x:=1;
while (Cmd_ObjIdx <> TabDefaultLux[x].LuxNumber) and ( x <= MAX_LUXNUM) do
	x := x + 1;	
end_while
if Cmd_ObjIdx = TabDefaultLux[x].LuxNumber and TabDefaultLux[x].Mode = 2 then	// Il crono vale solo per i lux con mode = 2

(* Process command *)
CASE Cmd_C OF

	1: (* GET PROFILE *)
		IF Cmd_CLen<>3 THEN
			Cmd_R:=4;
		ELSE
			(* Load profile *)
			CronEd.CN_Sel:=WORD_TO_BYTE(Cmd_ObjIdx);
				CronEd.CN_YSel:=Cmd_Buf[9];					//**
				CronEd.CN_YSel:=shl(CronEd.CN_YSel, 8);		//**
				CronEd.CN_YSel:=CronEd.CN_YSel+Cmd_Buf[8];	//**
				//Cmd_Buf_U16:=ADR(Cmd_Buf[8]); Sostituisco questa riga e la seguente con le 3 precedenti per little/big endian (**)
				//CronEd.CN_YSel:=Cmd_Buf_U16^;
			CronEd.PR_Sel:=Cmd_Buf[10];
			CronEd.PR_Load_Exe();
				for x:=0 to 95 do
					LocalSetpoint[x]:= int_to_word(CronEd.PR.Setpoint[x]);
					LocalSetpoint[x]:=rol(LocalSetpoint[x], 8); //Scambio byte per compatibilità con sistema wago little endian
				end_for
			(* Copy data *)
			Cmd_RLen:=192;
				//TxLen:=TxLen+RAWTOHEX(ADR(CronEd.PR.Setpoint),192,ADR(TxData[TxLen]));
				TxLen:=TxLen+RAWTOHEX(ADR(LocalSetpoint),192,ADR(TxData[TxLen]));
		END_IF

	2: (* SET PROFILE *)
		IF Cmd_CLen<>(3+192) THEN
			Cmd_R:=4;
		ELSE
			(* Save profile *)
			CronEd.CN_Sel:=WORD_TO_BYTE(Cmd_ObjIdx);
				CronEd.CN_YSel:=Cmd_Buf[9];					//**
				CronEd.CN_YSel:=shl(CronEd.CN_YSel, 8);		//**
				CronEd.CN_YSel:=CronEd.CN_YSel+Cmd_Buf[8];	//**
//				Cmd_Buf_U16:=ADR(Cmd_Buf[8]); Sostituisco questa riga e la seguente con le 3 precedenti per little/big endian (**)
//				CronEd.CN_YSel:=Cmd_Buf_U16^;
			CronEd.PR_Sel:=Cmd_Buf[10];
				MEMCPY(ADR(Cmd_Buf[11]),ADR(LocalSetpoint),192); //copio i dati in locale
				for x:=0 to 95 do
					LocalSetpoint[x]:=rol(LocalSetpoint[x], 8); //Scambio byte per compatibilità con sistema wago little endian
				end_for
				MEMCPY(ADR(LocalSetpoint),ADR(CronEd.PR.Setpoint),192); //copio i byte scambiati sopra nel setpoint del crono 
//				MEMCPY(ADR(Cmd_Buf[11]),ADR(CronEd.PR.Setpoint),192);
			CronEd.PR_Save_Exe();
		END_IF

	5: (* GET CALENDAR MONTH *)
		IF Cmd_CLen<>3 THEN
			Cmd_R:=4;
		ELSE
			(* Load calendar *)
			CronEd.CN_Sel:=WORD_TO_BYTE(Cmd_ObjIdx);
				CronEd.CN_YSel:=Cmd_Buf[9];					//**
				CronEd.CN_YSel:=shl(CronEd.CN_YSel, 8);		//**
				CronEd.CN_YSel:=CronEd.CN_YSel+Cmd_Buf[8];	//**
//				Cmd_Buf_U16:=ADR(Cmd_Buf[8]); Sostituisco questa riga e la seguente con le 3 precedenti per little/big endian (**)
//				CronEd.CN_YSel:=Cmd_Buf_U16^;
			CronEd.CA_Sel:=Cmd_Buf[10];
			CronEd.CA_Load_Exe();
			(* Copy data *)
			Cmd_RLen:=32;
			TxLen:=TxLen+RAWTOHEX(ADR(CronEd.CA.Profile),32,ADR(TxData[TxLen]));
		END_IF

	6: (* SET CALENDAR MONTH *)
		IF Cmd_CLen<>(3+32) THEN
			Cmd_R:=4;
		ELSE
			(* Save calendar *)
			CronEd.CN_Sel:=WORD_TO_BYTE(Cmd_ObjIdx);
				CronEd.CN_YSel:=Cmd_Buf[9];					//**
				CronEd.CN_YSel:=shl(CronEd.CN_YSel, 8);		//**
				CronEd.CN_YSel:=CronEd.CN_YSel+Cmd_Buf[8];	//**
//				Cmd_Buf_U16:=ADR(Cmd_Buf[8]); Sostituisco questa riga e la seguente con le 3 precedenti per little/big endian (**)
//				CronEd.CN_YSel:=Cmd_Buf_U16^;
			CronEd.CA_Sel:=Cmd_Buf[10];
			MEMCPY(ADR(Cmd_Buf[11]),ADR(CronEd.CA.Profile),32);
			CronEd.CA_Save_Exe();
		END_IF
		9: (* Active crono immediatly *)
			CronEd.CN_Sel:=WORD_TO_BYTE(Cmd_ObjIdx);
			for x:= 1 to CRON_MAX do
				if CRON[x].ID = CronEd.CN_Sel then
					CRON[x].InitOK:=FALSE;
				end_if
			end_for
	else
	Cmd_R:=3;
	end_case
else 
	Cmd_R:=2;
end_if
END_ACTION

ACTION Cmd_GRU:
(* Check index *)(*
IF Cmd_ObjIdx<>1 THEN
	Cmd_R:=2;
	RETURN;
END_IF

(* Process command *)
CASE Cmd_C OF

	1: (* GET CLIMATIC *)
		Cmd_RLen:=20;
		FOR i:=0 TO 4 DO
			j:=DINT_TO_INT(GRU01_Clima.Points[i].X);
			TxLen:=TxLen+RAWTOHEX(ADR(j),2,ADR(TxData[TxLen]));
			j:=DINT_TO_INT(GRU01_Clima.Points[i].Y);
			TxLen:=TxLen+RAWTOHEX(ADR(j),2,ADR(TxData[TxLen]));
		END_FOR

	2: (* SET CLIMATIC *)
		IF Cmd_CLen<>20 THEN
			Cmd_R:=4;
		ELSE
			FOR i:=0 TO 4 DO
				Cmd_Buf_INT:=ADR(Cmd_Buf[8+4*i]); j:=Cmd_Buf_INT^;
				GRU01_Clima.Points[i].X:=INT_TO_DINT(j);
				Cmd_Buf_INT:=ADR(Cmd_Buf[10+4*i]); j:=Cmd_Buf_INT^;
				GRU01_Clima.Points[i].Y:=INT_TO_DINT(j);
			END_FOR
		END_IF

ELSE
	Cmd_R:=3;
END_CASE
*);
END_ACTION

ACTION Cmd_PDC:
(* Check index *)(*
IF Cmd_ObjIdx<>1 THEN
	Cmd_R:=2;
	RETURN;
END_IF

(* Process command *)
CASE Cmd_C OF

	3: (* TRY REARM *)
		PDC01.Rearm:=TRUE;

ELSE
	Cmd_R:=3;
END_CASE
*);
END_ACTION

ACTION Cmd_SYS:
(* Check index *)
IF Cmd_ObjIdx<>0 THEN
	Cmd_R:=2;
	RETURN;
END_IF

(* Process command *)
CASE Cmd_C OF

	0: (* ECHO *)
		IF Cmd_CLen<>0 THEN
			TxLen:=0;
		END_IF

	1: (* LOG REQUEST *)
//		LogTrig();
		(*---------------------------------------------------------------*)
			Logger_Head();
		(*---------------------------------------------------------------*)
		FOR i := 1 TO MAX_LUXNUM DO	
			if LuxElement[i].ID <> 0
			then LuxElement[i].AddLogData(WORKINGTIME:=WORKINGTIME_n[i], POWERONCYCLES:=POWERONCYCLES_n[i],
							   ENERGYCOUNTER:=ENERGYCOUNTER_n[i], ENERGYCOUNTER_T:=ENERGYCOUNTER_T_n[i]);
			end_if
		END_FOR
		(*---------------------------------------------------------------*)
			Logger_Send();
		(*---------------------------------------------------------------*)

	2: (* REARM *)
		Sys.Warning:=FALSE;
		Sys.Alarm:=FALSE;
		Sys.AlarmStop:=FALSE;

	3: (* GET INFO1 *)
		Cmd_RLen:=6;
		Plant_SN_H:= Plant_SN and 16#FFFF0000;
		Plant_SN_L:= Plant_SN and 16#0000FFFF;
		Plant_SN_H:=shr(Plant_SN_H, 16);
		Plant_SN_H_W:=dword_to_word(Plant_SN_H);
		Plant_SN_H_W:=rol(Plant_SN_H_W, 8);
		Plant_SN_L_W:=dword_to_word(Plant_SN_L);
		Plant_SN_L_W:=rol(Plant_SN_L_W, 8);
		TxLen:=TxLen+RAWTOHEX(ADR(Plant_SN_H_W),2,ADR(TxData[TxLen]));
		TxLen:=TxLen+RAWTOHEX(ADR(Plant_SN_L_W),2,ADR(TxData[TxLen]));
		//TxLen:=TxLen+RAWTOHEX(ADR(Plant_SN),4,ADR(TxData[TxLen]));
		Plant_SW_VER:=rol(Plant_SW_VER, 8);
		TxLen:=TxLen+RAWTOHEX(ADR(Plant_SW_VER),2,ADR(TxData[TxLen]));

	14: (* Set data e ora *)
		Year:=byte_to_word(Cmd_Buf[8]); 
		Year:=SHL(Year,8);
		Year:=Year + byte_to_word(Cmd_Buf[9]); 
		Year:=rol(Year, 8);
		Month:=word_to_byte(Cmd_Buf[10]); 
		Day:=word_to_byte(Cmd_Buf[12]); 
		Hour:=word_to_byte(Cmd_Buf[14]); 
		minute:=word_to_byte(Cmd_Buf[16]); 
		Sec:=word_to_byte(Cmd_Buf[18]); 
(*	
		Year:=byte_to_word(Cmd_Buf[8]); 
		Year:=SHL(Year,8);
		Year:=Year + byte_to_word(Cmd_Buf[9]); 
		Month:=word_to_byte(Cmd_Buf[11]); 
		Day:=word_to_byte(Cmd_Buf[13]); 
		Hour:=word_to_byte(Cmd_Buf[15]); 
		minute:=word_to_byte(Cmd_Buf[17]); 
		Sec:=word_to_byte(Cmd_Buf[19]); 
*)
		DTStr := concat('DT#',word_to_string(Year));
		DTStr := concat(DTStr,'-');
		DTStr := concat(DTStr,byte_to_string(Month));
		DTStr := concat(DTStr,'-');
		DTStr := concat(DTStr,byte_to_string(Day));
		DTStr := concat(DTStr,'-');
		DTStr := concat(DTStr,byte_to_string(Hour));
		DTStr := concat(DTStr,':');
		DTStr := concat(DTStr,byte_to_string(minute));
		DTStr := concat(DTStr,':');
		DTStr := concat(DTStr,byte_to_string(Sec));
		DateTime:=string_to_dt(DTStr);
		Result:=SysRtcSetTime(DateTime);
ELSE
	Cmd_R:=3;
END_CASE
END_ACTION

ACTION Command:
(* Default response OK/NODATA *)
Cmd_R:=0;
Cmd_RLen:=0;
TxLen:=16;

(* Check object *)
CASE Cmd_Obj OF

	EO_SYS:
		Cmd_SYS();
(*
	EO_GRU:
		Cmd_GRU();

	EO_PDC:
		Cmd_PDC();

	EO_CAL:
		Cmd_CAL();
*)
	EO_CRON:
		Cmd_CRON();

	EO_LUX:
		Cmd_LUX();

ELSE
	Cmd_R:=1;
END_CASE

(* Generate response *)
IF TxLen>0 THEN
	Cmd_Obj:=rol(Cmd_Obj, 8); //Scambio byte per compatibilità con sistema wago little endian
	RAWTOHEX(ADR(Cmd_Obj)	,2,ADR(TxData[ 0]));
	Cmd_ObjIdx:=rol(Cmd_ObjIdx, 8); //Scambio byte per compatibilità con sistema wago little endian
	RAWTOHEX(ADR(Cmd_ObjIdx),2,ADR(TxData[ 4]));
	Cmd_R:=rol(Cmd_R, 8); //Scambio byte per compatibilità con sistema wago little endian
	RAWTOHEX(ADR(Cmd_R)		,2,ADR(TxData[ 8]));
	Cmd_RLen:=rol(Cmd_RLen, 8); //Scambio byte per compatibilità con sistema wago little endian
	RAWTOHEX(ADR(Cmd_RLen)	,2,ADR(TxData[12]));
	TxTrig:=TRUE;
END_IF
END_ACTION

ACTION Cmd_LUX:
(* Check index *)
if Cmd_ObjIdx<1 OR Cmd_ObjIdx>MAX_LUXNUM then
	Cmd_R:=2; //id del lux fuori range
	return;
end_if

x:=1;
while (Cmd_ObjIdx <> TabDefaultLux[x].LuxNumber) and ( x <= MAX_LUXNUM) do
	x := x + 1;	
end_while
if Cmd_ObjIdx = TabDefaultLux[x].LuxNumber then	
	(* Process command *)
	case Cmd_C of
	
		0:	(* Restore default functioning mode *)
		LuxElement[x].CTRL_MODE:=LuxElement[x].CTRL_MODE_backUp;
		LuxElement[x](WORKINGTIME:=WORKINGTIME_n[x],POWERONCYCLES:=POWERONCYCLES_n[x],
													ENERGYCOUNTER:=ENERGYCOUNTER_n[x], 
													ENERGYCOUNTER_T:=ENERGYCOUNTER_T_n[x],
													CtrlExton:=KEYON);

		1:	(* Reset statistic counter *)
		LuxElement[x].StatReset(WORKINGTIME:=WORKINGTIME_n[x],POWERONCYCLES:=POWERONCYCLES_n[x],
															ENERGYCOUNTER:=ENERGYCOUNTER_n[x], 
															ENERGYCOUNTER_T:=ENERGYCOUNTER_T_n[x],
															CtrlExton:=KEYON);
	
		2,3:	(* Switch On (command=2) or Off (command=3) lux *)
		case Cmd_C of
			2: (*switch a Manuale ON*)
			LuxElement[x].CTRL_MODE := 1; // Set to manuale ON
			LuxElement[x](WORKINGTIME:=WORKINGTIME_n[x],POWERONCYCLES:=POWERONCYCLES_n[x],
														ENERGYCOUNTER:=ENERGYCOUNTER_n[x], 
														ENERGYCOUNTER_T:=ENERGYCOUNTER_T_n[x],
														CtrlExton:=KEYON);
			3: (*switch a Manuale OFF*)
			LuxElement[x].CTRL_MODE := 0; // Set to manuale OFF
			LuxElement[x](WORKINGTIME:=WORKINGTIME_n[x],POWERONCYCLES:=POWERONCYCLES_n[x],
														ENERGYCOUNTER:=ENERGYCOUNTER_n[x], 
														ENERGYCOUNTER_T:=ENERGYCOUNTER_T_n[x],
														CtrlExton:=KEYON);
			
		end_case
		4: (* Modify timer value *)
		if TabDefaultLux[x].Mode = 03 then //la modifica ha senso per i lux a timer
			NewValueTimerH:=byte_to_word(Cmd_Buf[8]);
			NewValueTimerH:=SHL(NewValueTimerH,8); 
			NewValueTimerH:=NewValueTimerH+byte_to_word(Cmd_Buf[9]);
			NewValueTimerH:=rol(NewValueTimerH, 8);

			NewValueTimerL:=byte_to_word(Cmd_Buf[10]);
			NewValueTimerL:=SHL(NewValueTimerL,8); 
			NewValueTimerL:=NewValueTimerL+byte_to_word(Cmd_Buf[11]);
			NewValueTimerL:=rol(NewValueTimerL, 8);
			
			NewValueTimer:=word_to_dword(NewValueTimerH);			
			NewValueTimer:=SHL(NewValueTimer,16);
			NewValueTimer:=NewValueTimer+word_to_dword(NewValueTimerL);
			if NewValueTimer>4294966 then
				Cmd_R:=3; //Comando errato valore timer overflow		
			
(*
			NewValueTimer:=byte_to_dword(Cmd_Buf[8]);
			NewValueTimer:=SHL(NewValueTimer,8); 
			NewValueTimer:=NewValueTimer+byte_to_dword(Cmd_Buf[9]);
			NewValueTimer:=SHL(NewValueTimer,8); 
			NewValueTimer:=NewValueTimer+byte_to_dword(Cmd_Buf[10]);
			NewValueTimer:=SHL(NewValueTimer,8); 
			NewValueTimer:=NewValueTimer+byte_to_dword(Cmd_Buf[11]);
*)
			else
					TabLuxPsg[x].TimerOn := dword_to_time(NewValueTimer*1000);
				for x := 1 to MAX_LUXNUM do
					if LuxElement[x].ID = Cmd_ObjIdx
						then LuxElement[x].LuxTimer := dword_to_time(NewValueTimer*1000); //set del nuovo valore del timer del lux 	
					end_if
				end_for
			end_if
		else
			Cmd_R:=3; //Comando errato / non previsto
		end_if
		5:	(* get working mode*)
			Cmd_RLen:=2;
			ModeFromPlc:=LuxElement[x].CTRL_MODE;
			ModeFromPlc:=rol(ModeFromPlc, 8);
			TxLen:=TxLen+RAWTOHEX(ADR(ModeFromPlc),2,ADR(TxData[TxLen]));
//		6: (* Modify dimming value for timer control *)
//		7: (* Modify dimming value for key control *)
//		8: (* Modify start and stop orari di funzionamento dei lux a timer *)
	else
		Cmd_R:=3; //Comando errato / non previsto
	end_case
else
	Cmd_R:=2; //id del lux non presente in lista
end_if
END_ACTION

END_PROGRAM

// Utils Functions/HEXTORAW
FUNCTION HEXTORAW : WORD
VAR_INPUT
	pString		: POINTER TO BYTE;
	StringLen	: WORD;
	pData		: POINTER TO BYTE;
END_VAR
VAR
	xl: WORD;
	xi: WORD;
	xr: BYTE;
END_VAR

xl:=0;
xi:=0;

WHILE xi<StringLen DO

	IF pString^>=97 AND pString^<=102 THEN
		xr := pString^ - 87;
	ELSIF pString^>=65 AND pString^<=70 THEN
		xr := pString^ - 55;
	ELSIF pString^>=48 AND pString^<=57 THEN
		xr := pString^ - 48;
	ELSE
		xr := 16;
	END_IF

	IF xr<16 THEN
		IF (xi AND 1)=0 THEN
			pData^ := xr * 16;
		ELSE
			pData^ := pData^ + xr;
			pData := pData + 1;
			xl := xl + 1;
		END_IF
	END_IF

	xi := xi + 1;
	pString := pString + 1;

END_WHILE

HEXTORAW:=xl;

END_FUNCTION

// Utils Functions/TCPSERVER
FUNCTION_BLOCK TCPSERVER
(***********************************************************************************************************	*)
(* Version: 1.6                                    			          											*)
(* Date: 11.02.2011                                   					          							    *)
(***********************************************************************************************************	*)
(* WAGO Kontakttechnik GmbH Hansastr. 27 32423 Minden(Westf.)													*)
(* Tel. +0049 571/887-0 Fax. +0049 571/887-0																	*)
(* Author: VB																									*)
(***********************************************************************************************************	*)
(*Description:	A TCP server to read and write data													       		*)
(*Historie:																										*)
(*Version 1.6: 11.02.2011: Changes according to 750-880/881											 			*)
(*Version 1.5: 27.11.2008 Bugfix allow reuse port																*)
(*Version 1.4: 13.10.2008 Bugfix transmitting large data														*)
(*Version 1.3: 15.01.2007 Changes according to FW11																*)
(*Version 1.2: 09.03.2006 Changes for socket handle 0											       			*)
(*Version 1.1: 14.02.2005 Release																				*)
(***********************************************************************************************************	*)
VAR CONSTANT
	STATE_INIT     				 : BYTE:= 0;
	STATE_OPEN     				 : BYTE:= 1;
	STATE_TX       				 : BYTE:= 20;
	STATE_RX       				 : BYTE:= 30;
	STATE_CLOSE    				 : BYTE:= 40;
	STATE_ERROR_TRAP		 	 : BYTE:= 200;
END_VAR
VAR_INPUT
	xEnable    					: BOOL;	 (* Set TRUE to enable function block *)
	wPortNumber					: WORD;  (* Port *)
	tServerTimeOut				: TIME:=t#50s;
	ptSendData					: POINTER TO ARRAY[0..MAX_SEND_TCP_SERVER] OF BYTE;
	diSendCount					: DINT;
END_VAR
VAR_OUTPUT
	xClientConnected  			: BOOL:= FALSE;
	diError 					: DINT:= 0;
END_VAR
(* Status Codes -----------------------------------------
	16#8001 => No socket descriptor available 
	16#8002 => SysSockBind fails 
	16#8003 => SysSockListen fails 
	16#8004 => switching to none blocking mode fails
	16#8005 => SysSockClose() returns FALSE 
    16#8006 => SysSockConnect() fails
    16#8007 => SysSockSend() fails
	16#8008 => error state machine 
	16#8009 => timeout while waiting for data from server 
	16#0001 => server waiting for client to establish connection
------------------------------------------------------------*)
VAR_IN_OUT
	xStartSend					: BOOL;
	aReceiveBuffer				: ARRAY [0..MAX_RECEIVE_TCP_SERVER] OF BYTE;
	diReceiveCount				: DINT;
END_VAR

VAR
	m_State    					: BYTE:= 0;
	m_ReceiveBuffer				: ARRAY [0..MAX_RECEIVE_TCP_SERVER_SOCKET] OF BYTE;
	m_ServerSocket				: DINT:= SOCKET_INVALID;
	m_Socket					: DINT:= SOCKET_INVALID;
	m_AddressInfo				: SOCKADDRESS;
	m_BytesReceived				: DINT;
	m_diReturn					: DINT;
	m_xReturn					: BOOL;
	m_SizeSockadr				: DWORD;
	m_ConnectionWatchdog		: TON;
	m_Flags						: DINT;
	m_NoneBlocking   			: DINT:= 1;
	m_Blocking   				: DINT:= 0;
	i							: INT;
	m_count						: DINT;
	diOption					: DINT := 1;
	on: DINT;
	errorCode					: DINT;
	errorCodeLenght				: dint;
	xResultErrCode				: bool;
END_VAR

IF xEnable THEN
	CASE m_State OF
		STATE_INIT:
			(* Create Socket *)
			m_ServerSocket:= SysSockCreate( SOCKET_AF_INET, SOCKET_STREAM, 0);
			IF m_ServerSocket = SOCKET_INVALID THEN
				(* *)
				diError:= 16#8001;
				m_State:= STATE_ERROR_TRAP;
				RETURN;
			ELSE
				;
			END_IF
			(* Address bindings *)
			(********************)
			on:=1;
			SysSockSetOption( m_ServerSocket, SOCKET_SOL, SOCKET_SO_REUSEADDR, ADR(on), SIZEOF(on) );

			m_AddressInfo.sin_family:= SOCKET_AF_INET;
			m_AddressInfo.sin_port  := SysSockHtons( wPortNumber);
			m_AddressInfo.sin_addr  := SOCKET_INADDR_ANY;
			IF NOT SysSockBind( m_ServerSocket, ADR(m_AddressInfo), SIZEOF(m_AddressInfo)) THEN
				diError:= 16#8002;
				m_State:= STATE_ERROR_TRAP;
				RETURN;
			END_IF
			(* Wait for connections *)
			(************************)
			IF NOT SysSockListen( m_ServerSocket, 1) THEN
				diError:= 16#8003;
				m_State:= STATE_ERROR_TRAP;
			END_IF

			(* Puts SOCKET in NonBlocking mode *)
			m_diReturn:= SysSockIoctl( m_ServerSocket, SOCKET_FIONBIO, ADR(m_NoneBlocking));

			m_State:= STATE_OPEN;


		STATE_OPEN: 	(* Waiting for incomming connection *)
				m_SizeSockadr:=SIZEOF(m_AddressInfo);
				m_Socket:= SysSockAccept( m_ServerSocket, ADR(m_AddressInfo), ADR(m_SizeSockadr));
				diError:=State_open;
				IF m_Socket <> SOCKET_INVALID THEN
					xClientConnected:=TRUE;
					(*Set Push-Bit:new V1.5*)
				(*	IF ADR(%MW0)=16#30000000  OR ADR(%MW0)=16#20000000 THEN (*841 or 881*)
						SysSockSetOption(
							diSocket:=m_Socket,
							diLevel:=6,
							diOption:=SOCKET_TCP_NODELAY,
							pOptionValue:=ADR(diOption),
							diOptionLength:=SIZEOF(diOption));
					ELSE
							;
					END_IF *)
					SysSockIoctl( m_Socket, SOCKET_FIONBIO, ADR(m_NoneBlocking));
					m_State:= STATE_RX;
					diError:=0;
				END_IF

		STATE_RX:
					errorCodeLenght:=sizeof(errorCode);
					xResultErrCode:=SysSockGetOption(m_Socket,  SOCKET_SOL, SOCKET_SO_KEEPALIVE, adr(errorCode), adr(errorCodeLenght));
					m_BytesReceived:= SysSockRecv( m_Socket, ADR(m_ReceiveBuffer), SIZEOF(m_ReceiveBuffer), 0);
					CASE m_BytesReceived OF
					-1:(*no data available or error occured*)
						m_ConnectionWatchdog(IN:=TRUE , PT:=T#200ms);	//tServerTimeOut );
						IF m_connectionWatchdog.Q THEN
							m_State:= STATE_CLOSE;
							m_ConnectionWatchdog(IN:=FALSE);(*reset connection watchdog*)
							diError := 16#8009;
						END_IF
					0:(* socket was "gracefully closed"  *)
						m_State:= STATE_CLOSE;
						diError := 16#8003;
					ELSE
						(* Copy received data into receive buffer *)
						(********************************)
						FOR i:= 0 TO DINT_TO_INT(m_BytesReceived	)-1 DO
							aReceiveBuffer[diReceiveCount]:= m_ReceiveBuffer[i];
							diReceiveCount:=(diReceiveCount+1) MOD SIZEOF(aReceiveBuffer);
						END_FOR

						m_ConnectionWatchdog(IN:=FALSE);(*reset connection watchdog*)
					END_CASE

				(*send data*)
				IF xStartSend	 THEN
					m_State := STATE_TX;
				END_IF

	STATE_TX:	 (* send TCP-message *)
		m_diReturn := SysSockSend(diSocket := m_Socket,
								  pbyBuffer := ADR(ptSendData^[m_count]),(*geändert V1.4 bisher: [0] *)
								  diBufferSize := diSendCount-m_count,
								  diFlags :=m_Flags);
		CASE m_diReturn OF
		-1:	(* ERROR or data could not yet be send (V1.3 due to new FW11) *)
			m_ConnectionWatchdog(IN:=TRUE , PT:=tServerTimeOut );
			IF m_connectionWatchdog.Q THEN
				m_State:= STATE_CLOSE;
				m_ConnectionWatchdog(IN:=FALSE);(*reset connection watchdog*)
				diError := 16#8007;
			END_IF
		0: (* socket was "gracefully closed"  *)
			m_State := STATE_CLOSE;
			diError := 16#8003;
		ELSE (* succesful *)
			m_count:=m_count+m_diReturn;
			IF m_count>=diSendCount THEN
				diError := 16#0000;
				m_State := STATE_RX;
				m_count:=0;
				xStartSend:=FALSE;
			END_IF
			m_ConnectionWatchdog(IN:=FALSE);(*reset connection watchdog*)
		END_CASE


		STATE_CLOSE:	(* Close the server *)

	(*	IF ADR(%MW0)=16#30000000  OR ADR(%MW0)=16#20000000 THEN (*841 or 881*)
			;
		ELSE
			IF m_Socket>=0 THEN
				SysSockShutdown(m_Socket, 0);;(*870*)
			END_IF
		END_IF  *)
		IF m_Socket>=0 THEN
			SysSockClose( m_Socket);
		END_IF
		xClientConnected:= FALSE;
		m_State:= STATE_OPEN; (* Try to open the server again *)
		m_ConnectionWatchdog(IN:=FALSE);(*reset connection watchdog*)

		STATE_ERROR_TRAP: (* Error Read/Write socket  *)
			m_State:= STATE_ERROR_TRAP;

	ELSE  (* Bad FSM code trap  *)
			m_State:= STATE_ERROR_TRAP;
			diError:= 16#8008;
	END_CASE;
ELSE
	IF m_State <> STATE_INIT THEN
	(*	IF ADR(%MW0)=16#30000000  OR ADR(%MW0)=16#20000000 THEN (*841 or 881*)
			;
		ELSE
			IF m_Socket>=0 THEN
				SysSockShutdown(m_Socket, 0);;(*870*)
			END_IF
		END_IF *)
		IF m_Socket>=0 THEN
			SysSockClose( m_Socket);
		END_IF
	(*	IF ADR(%MW0)=16#30000000  OR ADR(%MW0)=16#20000000 THEN (*841 or 881*)
			;
		ELSE
			IF m_ServerSocket>=0 THEN
				SysSockShutdown(m_ServerSocket, 0);;(*870*)
			END_IF
		END_IF  *)
		IF m_ServerSocket>=0 THEN
			SysSockClose( m_ServerSocket);
		END_IF
		xClientConnected:= FALSE;
		diError:= 0;
		m_State:= STATE_init; (* Try to open the server again *)
		m_ConnectionWatchdog(IN:=FALSE);(*reset connection watchdog*)
	END_IF
END_IF

END_FUNCTION_BLOCK

// Utils Functions/RAWTOHEX
FUNCTION RAWTOHEX : WORD
VAR_INPUT
	pData: POINTER TO BYTE;
	DataLen: WORD;
	pString: POINTER TO BYTE;
END_VAR
VAR
	xl: WORD;
END_VAR

xl:=0;

WHILE DataLen>0 DO

	pString^ := (pData^ / 16#10) + 48 + (((pData^ / 16#10)/10)*7);
	pString:=pString+1;
	pString^ := (pData^ AND 16#0F)  + 48 + (((pData^ AND 16#0F)/10)*7);
	pString:=pString+1;
	pData:=pData+1;
	DataLen:=DataLen-1;
	xl:=xl+2;

END_WHILE

(*pString^:=0;*)

RAWTOHEX:=xl;

END_FUNCTION

// TCP_Logger/LogTrig
FUNCTION LogTrig : BOOL
VAR
	s1 		: STRING(255);	//STRING(160);
	i, j, k	: word;
END_VAR

(*---------------------------------------------------------------*)
	Logger_Head();
(*---------------------------------------------------------------*)
case enSelect of
	Sel_PSG: (* Log PSG *)

for i := 1 TO PSG_MAXNUM DO	
	if PSG[i].ID <> 0
	then PSG[i].AddLogData(NumTransition:=PsgCounter[i]);	//PSG[i].AddLogData(NumTransition:=PsgCounter[PSG[i].ID]);
 	end_if
END_FOR
		enSelect:=Sel_LUX;
		
	Sel_LUX: (* Log LUXM *)
		
FOR i := 1 TO MAX_LUXNUM DO	
	if LuxElement[i].ID <> 0
	then LuxElement[i].AddLogData(WORKINGTIME:=WORKINGTIME_n[i], POWERONCYCLES:=POWERONCYCLES_n[i],
					   ENERGYCOUNTER:=ENERGYCOUNTER_n[i], ENERGYCOUNTER_T:=ENERGYCOUNTER_T_n[i]);
 	end_if
END_FOR
		enSelect:=Sel_CRON;
	Sel_CRON: (* Log CRON *)

FOR i := 1 TO CRON_MAX DO
	if CRON[i].ID <> 0
		then CRON[i].AddLogData(SET_POINT:=CRON[i].SetPoint, STAT_LOG:=CRON[i].Status_Log);
	end_if
END_FOR

		enSelect:=Sel_END;
END_CASE
(* Log LUXM *)
	(* 
FOR i := 1 TO MAX_LUXNUM DO	
	if LuxElement[i].ID <> 0
	then LuxElement[i].AddLogData(WORKINGTIME:=WORKINGTIME_n[i], POWERONCYCLES:=POWERONCYCLES_n[i],
					   ENERGYCOUNTER:=ENERGYCOUNTER_n[i], ENERGYCOUNTER_T:=ENERGYCOUNTER_T_n[i]);
 	end_if
END_FOR
 *)

(*---------------------------------------------------------------*)
	Logger_Send();
(*---------------------------------------------------------------*)

END_FUNCTION

// Utils Functions/TestAsi_FB
FUNCTION_BLOCK TestAsi_FB
VAR_INPUT
END_VAR
VAR_OUTPUT
END_VAR
VAR
	TTestOut: tof
;
	iCounter0: INT := 0;
	TrigH:	BOOL;
	rTrigger: R_TRIG;
END_VAR

(*
TTestOut(IN:=NOT TTestOut.Q,PT:=T#5S);
IF TTestOut.Q AND LUXM_46 = FALSE
THEN
	LUXM_46:=TRUE;	
	ELSE
		IF NOT TTestOut.Q
			THEN
				LUXM_46 := FALSE;
		END_IF
END_IF
IF 	LUXST_46 THEN
	IF iCounter0 < 65535 THEN
		iCounter0:=iCounter0+1;	
	END_IF
END_IF
*)
//rTrigger(CLK:=PSG89_IN);
//TTestOut(IN:=NOT PSG89_IN ,PT:=T#5S);
//IF rTrigger.q THEN
 	//TTestOut(IN:=rTrigger.q ,PT:=T#5S);
//END_IF
(*
IF TTestOut.Q THEN 
	LUXM_46:=TRUE;	
	ELSE
		LUXM_46:=FALSE;	
END_IF
*)
(*
IF 	Asi_in0901 THEN
	IF iCounter1 < 65535 THEN
		iCounter1:=iCounter1+1;	
	END_IF

END_IF

IF 	Asi_in0902 THEN
	IF iCounter2 < 65535 THEN
		iCounter2:=iCounter2+1;	
	END_IF
END_IF

IF 	Asi_in0903 THEN
	IF iCounter3 < 65535 THEN
		iCounter3:=iCounter3+1;	
	END_IF

END_IF
*)

END_FUNCTION_BLOCK

// Utils Functions/OpenFiles_ASI_PSG_FB
//Esegue la lettura del file x_ASI_PSG.txt per poi configurare le tabelle ASI_1 e ASI_2 di associazione tra passaggi e segnali di input 
FUNCTION_BLOCK OpenFiles_ASI_PSG_FB
VAR_INPUT
	//sFileName : STRING;
END_VAR
VAR_OUTPUT
	Message		: STRING;
END_VAR
VAR
	hMode		: ACCESS_MODE;
	hFile		: RTS_IEC_HANDLE;
	hRes		: RTS_IEC_RESULT;
	bList		: ARRAY [0..15] OF BYTE;
	i			: DWORD; //Dim max file: 2^32 byte
	j			: BYTE; //Indice dell'array bList
	k			: BYTE; //Indice tabella ASI 2^8 = 256
	xwDimFile	: LWORD;
	bChar		: BYTE;
	sFileName 	: STRING;
END_VAR

(* Create current filename 'yyyyCRnn.DAT' *)
//sFileName:=CONCAT(ConfPath,WORD_TO_STRING('2ASI_LUX.txt'));
//sFileName:=CONCAT(STR1:=sFileName, STR2:='CR');
//IF CN_Sel<10 THEN
//sFileName:=CONCAT(STR1:=sFileName, STR2:='0');
//END_IF
//sFileName:=CONCAT(STR1:=sFileName, STR2:=BYTE_TO_STRING(CN_Sel));
//sFileName:=CONCAT(STR1:=sFileName, STR2:='.DAT');
//sFileName:='/media/sd/2015CR01.DAT';	//2_ASI_LUX.txt';
(* Check file version and size! *)
(* ... *)
Message:='';
(* Open data file *)
sFileName:=CONCAT(STR1:=MapConf_Path, STR2:=PLC_ID);
sFileName:=CONCAT(STR1:=sFileName, STR2:=AsiPsg_FileName);
hFile:=SysFileOpen(sFileName,AM_READ,ADR(hRes));

(* File not found *)
IF hFile=RTS_INVALID_HANDLE THEN
	Message:='File not found';
	RETURN;
END_IF

(* Close file *)
SysFileClose(hFile);

(* Open data file *)
i:=0; //indice di scorrimento del file
j:=0; //indice di scorrimento dell'array dove viene momentaneamente memorizzata la riga prima del ;
k:=0; //indice della tabella di mappatura ASI
hFile:=SysFileOpen(sFileName,hMode,ADR(hRes));
//-------------- MODIFICA START --------------------
	SysFileSetPos(hFile, i);	
	SysFileRead(hFile, ADR(bList[j]), 1, ADR(hRes));
//-------------- MODIFICA END --------------------
WHILE SysFileEOF(hFile)<> 0 DO
//	SysFileSetPos(hFile, i);	
//	SysFileRead(hFile, ADR(bList[j]), 1, ADR(hRes));
	IF bList[j] = 16#2F  // se trovo '/'
		THEN 
			SysFileSetPos(hFile, i+1);	
			SysFileRead(hFile, ADR(bList[j+1]), 1, ADR(hRes));
			IF bList[j+1] = 16#2F  // se trovo ancora '/'
				THEN 
					WHILE  bList[j]<> 16#0D DO
						i := i+1;
						SysFileSetPos(hFile, i);	
						SysFileRead(hFile, ADR(bList[j]), 1, ADR(hRes));
					END_WHILE	
					i := i+1;
					SysFileSetPos(hFile, i);	
					SysFileRead(hFile, ADR(bList[j]), 1, ADR(hRes));
					IF bList[j] = 16#0A
						THEN 
							i := i+1;
							j := 0;
							SysFileSetPos(hFile, i);	
							SysFileRead(hFile, ADR(bList[j]), 1, ADR(hRes)); //leggo il primo carattere della nuova riga
						ELSE 
							Message:='Errore 0D 0A';
							RETURN;
					END_IF
				ELSE 
					Message:='Errore //';
					RETURN;
			END_IF
	END_IF
	IF bList[j] <> 16#3B //finchè non trovo ;
		THEN 
			i:=i+1;
			j:=j+1;	
		ELSE
			i:=i+3; //Se trovo ; inizio a salvare i dati della riga letta in TabAsiPsg[k]....
			j:=0;
			k:=k+1;
			TabAsiPsg[k].Asi1_2 := (bList[0]-16#30); //memorizzo se asi 1 o asi 2
			IF 	bList[4] = 16#41	//Se contiene il carattere A
				THEN TabAsiPsg[k].A_B := ASI_A;
				ELSE TabAsiPsg[k].A_B := ASI_B;
			END_IF	
			TabAsiPsg[k].Address :=  (bList[2]-16#30)*10 + (bList[3]-16#30); //memorizzo indirizzo
			TabAsiPsg[k].bit_psg[bList[6]-16#30] := (bList[8]-16#30)*100 + (bList[9]-16#30)*10 + (bList[10]-16#30); //memorizzo il passaggio associato 
			//TabAsiPsg[k].PSG := (bList[8]-16#30)*100 + (bList[9]-16#30)*10 + (bList[10]-16#30); //memorizzo il passaggio associato
			IF 	(k> 1) AND (TabAsiPsg[k].Asi1_2 = TabAsiPsg[k-1].Asi1_2) AND (TabAsiPsg[k].A_B = TabAsiPsg[k-1].A_B) AND (TabAsiPsg[k].Address = TabAsiPsg[k-1].Address)
				THEN //memorizzo il passaggio associato nella struttura k-1 perchè di uguale indirizzo
					TabAsiPsg[k-1].bit_psg[bList[6]-16#30] := (bList[8]-16#30)*100 + (bList[9]-16#30)*10 + (bList[10]-16#30);  
					TabAsiPsg[k].Asi1_2 := 0;	//pulisco l'array
					TabAsiPsg[k].A_B := 0;	//pulisco l'array
					TabAsiPsg[k].Address := 0;	//pulisco l'array
					TabAsiPsg[k].bit_psg[bList[6]-16#30] := 0;	//pulisco l'array
					k := k-1;	//riposiziono il contatore
			END_IF
			(*		
			CASE bList[0] OF
			16#31:
				IF 	bList[4] = 16#41	//Se contiene il carattere A
					THEN TabASI1[k].A_B := ASI_A;
					ELSE TabASI1[k].A_B := ASI_B;
				END_IF		
				TabASI1[k].Address :=  (bList[2]-16#30)*10 + (bList[3]-16#30);
				TabASI1[k].Bit_address := bList[6]-16#30;
				TabASI1[k].PSG := (bList[8]-16#30)*100 + (bList[9]-16#30)*10 + (bList[10]-16#30);
				
			16#32:
				IF 	bList[4] = 16#41	//Se contiene il carattere A
					THEN TabASI2[k].A_B := ASI_A;
					ELSE TabASI2[k].A_B := ASI_B;
				END_IF		
				TabASI2[k].Address :=  (bList[2]-16#30)*10 + (bList[3]-16#30);
				TabASI2[k].Bit_address := bList[6]-16#30;
				TabASI2[k].PSG := (bList[8]-16#30)*100 + (bList[9]-16#30)*10 + (bList[10]-16#30);
		END_CASE 
			CASE bList[0] OF
			16#31:
				IF 	bList[4] = 16#41	//Se contiene il carattere A
					THEN TabASI1AB_FromFile[1] := ASI_A;
					ELSE TabASI1AB_FromFile[1] := ASI_B;
				END_IF		
				TabASI1Add_FromFile[1] :=  (bList[2]-16#30)*10 + (bList[3]-16#30);
				TabASI1BitAdd_FromFile[1] := bList[6]-16#30;
				TabASI1PSG_FromFile[1] := (bList[8]-16#30)*100 + (bList[9]-16#30)*10 + (bList[10]-16#30);
			16#32:
				IF 	bList[4] = 16#41	//Se contiene il carattere A
					THEN TabASI2AB_FromFile[1] := ASI_A;
					ELSE TabASI2AB_FromFile[1] := ASI_B;
				END_IF		
				TabASI2Add_FromFile[1] :=  (bList[2]-16#30)*10 + (bList[3]-16#30);
				TabASI2BitAdd_FromFile[1] := bList[6]-16#30;
				TabASI2PSG_FromFile[1] := (bList[8]-16#30)*100 + (bList[9]-16#30)*10 + (bList[10]-16#30);
		END_CASE *)
	END_IF	
//-------------- MODIFICA START --------------------
	SysFileSetPos(hFile, i);	
	SysFileRead(hFile, ADR(bList[j]), 1, ADR(hRes));
//-------------- MODIFICA END --------------------
END_WHILE
if SysFileEOF(hFile) = 0 
	then Message:='Reading ASI_Psg File: OK';
end_if
//xwDimFile:=SysFileGetSize(sFileName,ADR(hRes));
(* Close file *)
SysFileClose(hFile);

END_FUNCTION_BLOCK

// Utils Functions/OpenFiles_ASI_LUX_FB
//Esegue la lettura del file x_ASI_LUX.txt per poi configurare le tabelle ASI_1 e ASI_2 di associazione tra LUX e segnali di output 
FUNCTION_BLOCK OpenFiles_ASI_LUX_FB
VAR_INPUT
END_VAR
VAR_OUTPUT
	Message		: STRING;
END_VAR
VAR
	hMode		: ACCESS_MODE;
	hFile		: RTS_IEC_HANDLE;
	hRes		: RTS_IEC_RESULT;
	bList		: ARRAY [0..15] OF BYTE;
	i			: DWORD;
	j			: DWORD;
	k			: byte;
	xwDimFile	: LWORD;
	bChar		: BYTE;
	sFileName 	: STRING;
END_VAR

Message:='';
(* Open data file *)
sFileName:=CONCAT(STR1:=MapConf_Path, STR2:=PLC_ID);
sFileName:=CONCAT(STR1:=sFileName, STR2:=AsiLux_FileName);
hFile:=SysFileOpen(sFileName,AM_READ,ADR(hRes));

(* File not found *)
IF hFile=RTS_INVALID_HANDLE THEN
	Message:='File not found';
	RETURN;
END_IF

(* Close file *)
SysFileClose(hFile);

(* Open data file *)
i:=0;
j:=0;
k:=0;
hFile:=SysFileOpen(sFileName,hMode,ADR(hRes));
//-------------- MODIFICA START --------------------
	SysFileSetPos(hFile, i);	
	SysFileRead(hFile, ADR(bList[j]), 1, ADR(hRes));
//-------------- MODIFICA END --------------------
WHILE SysFileEOF(hFile)<> 0 DO
//	SysFileSetPos(hFile, i);	
//	SysFileRead(hFile, ADR(bList[j]), 1, ADR(hRes));
	IF bList[j] = 16#2F  // se trovo '/'
		THEN 
			SysFileSetPos(hFile, i+1);	
			SysFileRead(hFile, ADR(bList[j+1]), 1, ADR(hRes));
			IF bList[j+1] = 16#2F  // se trovo ancora '/'
				THEN 
					WHILE  bList[j]<> 16#0D DO
						i := i+1;
						SysFileSetPos(hFile, i);	
						SysFileRead(hFile, ADR(bList[j]), 1, ADR(hRes));
					END_WHILE	
					i := i+1;
					SysFileSetPos(hFile, i);	
					SysFileRead(hFile, ADR(bList[j]), 1, ADR(hRes));
					IF bList[j] = 16#0A
						THEN 
							i := i+1;
							j := 0;
							SysFileSetPos(hFile, i);	
							SysFileRead(hFile, ADR(bList[j]), 1, ADR(hRes)); //leggo il primo carattere della nuova riga
						ELSE 
							Message:='Errore 0D 0A';
							RETURN;
					END_IF
				ELSE 
					Message:='Errore //';
					RETURN;
			END_IF
	END_IF
	IF bList[j] <> 16#3B //finchè non trovo ;
		THEN 
			i:=i+1;
			j:=j+1;	
		ELSE
			i:=i+3; //Se trovo ; inizio a salvare i dati della riga letta in TabASILux[k]....
			j:=0;
			k:=k+1;
			TabASILux[k].Asi1_2 := (bList[0]-16#30); //memorizzo se asi 1 o asi 2
			IF 	bList[4] = 16#41	//Se contiene il carattere A
				THEN TabASILux[k].A_B := ASI_A;
				ELSE TabASILux[k].A_B := ASI_B;
			END_IF		
			TabASILux[k].Address :=  (bList[2]-16#30)*10 + (bList[3]-16#30); //memorizzo indirizzo
			TabASILux[k].bit_lux[bList[6]-16#30] := (bList[8]-16#30)*100 + (bList[9]-16#30)*10 + (bList[10]-16#30); //memorizzo il lux associato 
			IF 	(k> 1) AND (TabASILux[k].Asi1_2 = TabASILux[k-1].Asi1_2) AND (TabASILux[k].A_B = TabASILux[k-1].A_B) AND (TabASILux[k].Address = TabASILux[k-1].Address)
				THEN //memorizzo il passaggio associato nella struttura k-1 perchè di uguale indirizzo
					TabASILux[k-1].bit_lux[bList[6]-16#30] := (bList[8]-16#30)*100 + (bList[9]-16#30)*10 + (bList[10]-16#30);  
					TabASILux[k].Asi1_2 := 0;	//pulisco l'array
					TabASILux[k].A_B := 0;	//pulisco l'array
					TabASILux[k].Address := 0;	//pulisco l'array
					TabASILux[k].bit_lux[bList[6]-16#30] := 0;	//pulisco l'array
					k := k-1;	//riposiziono il contatore
			END_IF
			
//			TabASILux[k].Address :=  (bList[2]-16#30)*10 + (bList[3]-16#30); //memorizzo indirizzo
//			TabASILux[k].Bit_address := bList[6]-16#30;		//memorizzo il bit
//			TabASILux[k].LUX := (bList[8]-16#30)*100 + (bList[9]-16#30)*10 + (bList[10]-16#30); //memorizzo il passaggio associato
	END_IF	
//-------------- MODIFICA START --------------------
	SysFileSetPos(hFile, i);	
	SysFileRead(hFile, ADR(bList[j]), 1, ADR(hRes));
//-------------- MODIFICA END --------------------
END_WHILE
if SysFileEOF(hFile) = 0 
	then Message:='Reading ASI_Lux File: OK';
end_if
(* Close file *)
SysFileClose(hFile);

END_FUNCTION_BLOCK

// Utils Functions/OpenFiles_LUX_PSG_FB
//Esegue la lettura del file x_AUT_LUX_PSG.txt per poi configurare le associazione tra passaggi e lux corrispondenti
FUNCTION_BLOCK OpenFiles_LUX_PSG_FB
VAR_INPUT
	//sFileName : STRING;
END_VAR
VAR_OUTPUT
	Message		: STRING;
END_VAR
VAR
	hMode		: ACCESS_MODE;
	hFile		: RTS_IEC_HANDLE;
	hRes		: RTS_IEC_RESULT;
	bList		: ARRAY [0..79] OF BYTE;
	i			: DWORD; //Dim max file: 2^32 byte
	j			: BYTE; //Indice dell'array bList
	k			: BYTE; //Indice tabella ASI 2^8 = 256
	x			: BYTE;
	xwDimFile	: LWORD;
	bChar		: BYTE;
	sFileName, TodString 	: STRING;
	TimerValue				: WORD;
	psgCount, local_x		: BYTE;

	
END_VAR

(* Create current filename 'yyyyCRnn.DAT' *)
//sFileName:=CONCAT(ConfPath,WORD_TO_STRING('2ASI_LUX.txt'));
//sFileName:=CONCAT(STR1:=sFileName, STR2:='CR');
//IF CN_Sel<10 THEN
//sFileName:=CONCAT(STR1:=sFileName, STR2:='0');
//END_IF
//sFileName:=CONCAT(STR1:=sFileName, STR2:=BYTE_TO_STRING(CN_Sel));
//sFileName:=CONCAT(STR1:=sFileName, STR2:='.DAT');
//sFileName:='/media/sd/2015CR01.DAT';	//2_ASI_LUX.txt';
(* Check file version and size! *)
(* ... *)
Message:='';
(* Open data file *)
sFileName:=CONCAT(STR1:=MapConf_Path, STR2:=PLC_ID);
sFileName:=CONCAT(STR1:=sFileName, STR2:=LuxPsg_FileName);
hFile:=SysFileOpen(sFileName,AM_READ,ADR(hRes));

(* File not found *)
IF hFile=RTS_INVALID_HANDLE THEN
	Message:='File not found';
	RETURN;
END_IF

(* Close file *)
SysFileClose(hFile);

(* Open data file *)
i:=0; //indice di scorrimento del file
j:=0; //indice di scorrimento dell'array dove viene momentaneamente memorizzata la riga prima del ;
k:=0; //indice della tabella di mappatura ASI
hFile:=SysFileOpen(sFileName,hMode,ADR(hRes));
//-------------- MODIFICA START --------------------
	SysFileSetPos(hFile, i);	
	SysFileRead(hFile, ADR(bList[j]), 1, ADR(hRes));
//-------------- MODIFICA END --------------------
WHILE SysFileEOF(hFile)<> 0 DO
//	SysFileSetPos(hFile, i);	
//	SysFileRead(hFile, ADR(bList[j]), 1, ADR(hRes));
	IF bList[j] = 16#2F  // se trovo '/'
		THEN 
			SysFileSetPos(hFile, i+1);	
			SysFileRead(hFile, ADR(bList[j+1]), 1, ADR(hRes));
			IF bList[j+1] = 16#2F  // se trovo ancora '/'
				THEN 
					WHILE  bList[j]<> 16#0D DO
						i := i+1;
						SysFileSetPos(hFile, i);	
						SysFileRead(hFile, ADR(bList[j]), 1, ADR(hRes));
					END_WHILE	
					i := i+1;
					SysFileSetPos(hFile, i);	
					SysFileRead(hFile, ADR(bList[j]), 1, ADR(hRes));
					IF bList[j] = 16#0A
						THEN 
							i := i+1;
							j := 0;
							SysFileSetPos(hFile, i);	
							SysFileRead(hFile, ADR(bList[j]), 1, ADR(hRes)); //leggo il primo carattere della nuova riga
						ELSE 
							Message:='Errore 0D 0A';
							RETURN;
					END_IF
				ELSE 
					Message:='Errore //';
					RETURN;
			END_IF
	END_IF
	IF bList[j] <> 16#3B //finchè non trovo ;
		THEN 
			i:=i+1;
			j:=j+1;	
		ELSE
			i:=i+3; //Se trovo ; inizio a salvare i dati della riga letta in TabLuxPsg[k]....
			j:=0;
			k:=k+1;
			x:=0;
			WHILE (bList[x]<>16#3B) DO  //bList[x]<>';'
				CASE (bList[x]) OF
				(*L*)16#4C: TabLuxPsg[k].LuxId := ((bList[x+1]-16#30)*100+(bList[x+2]-16#30)*10+(bList[x+3]-16#30));
				(*T*)16#54: TimerValue := ((bList[x+1]-16#30)*10000+(bList[x+2]-16#30)*1000+(bList[x+3]-16#30)*100 +(bList[x+4]-16#30)*10 +(bList[x+5]-16#30));
							TabLuxPsg[k].TimerOn := DWORD_TO_TIME(TimerValue*1000); //(bList[x+1]-16#30)*10+(bList[x+2]-16#30);
				(*O*)16#4F: TodString := concat('TOD#',BYTE_TO_STRING(bList[x+1]-16#30));
							TodString := concat(TodString,BYTE_TO_STRING(bList[x+2]-16#30));
							TodString := concat(TodString,':');
							TodString := concat(TodString,BYTE_TO_STRING((bList[x+4]-16#30)));
							TodString := concat(TodString,BYTE_TO_STRING((bList[x+5]-16#30)));
							TabLuxPsg[k].h_Start := STRING_TO_TOD(TodString);  //TabLuxPsg[k].TimerOn := (bList[x+1]-16#30)*10+(bList[x+2]-16#30);
							TodString := concat('TOD#',BYTE_TO_STRING(bList[x+7]-16#30));
							TodString := concat(TodString,BYTE_TO_STRING(bList[x+8]-16#30));
							TodString := concat(TodString,':');
							TodString := concat(TodString,BYTE_TO_STRING((bList[x+10]-16#30)));
							TodString := concat(TodString,BYTE_TO_STRING((bList[x+11]-16#30)));
							TabLuxPsg[k].h_End := STRING_TO_TOD(TodString); 
				(*S*)16#53:	TabLuxPsg[k].scaIdUnit := (bList[x+1]-16#30)*10+(bList[x+2]-16#30);		
							TabLuxPsg[k].scaIdDec := (bList[x+4]-16#30)*10+(bList[x+5]-16#30);	
				(*S*)16#50:	local_x := x;
							FOR psgCount := 0 TO MAX_PSGLIST BY 1 DO //Leggo un massimo di 10 passaggi associati a quel lux
								IF (bList[local_x] <> 16#3B) //Se trovo ; termino la lettura dei passaggi e vado alla riga successiva del file
									THEN
										TabLuxPsg[k].PSG_list[psgCount] := (bList[local_x+1]-16#30)*100+(bList[local_x+2]-16#30)*10+(bList[local_x+3]-16#30);
										local_x:=local_x+4;
									ELSE 
										//x:= 0; //ho terminato di leggere il contenuto di bList[] quindi resetto l'indice e esco. Vado a leggere la riga successiva del file 
										EXIT;
								END_IF
							END_FOR;		
				END_CASE
				x:=x+1;
			END_WHILE
	END_IF	
//-------------- MODIFICA START --------------------
	SysFileSetPos(hFile, i);	
	SysFileRead(hFile, ADR(bList[j]), 1, ADR(hRes));
//-------------- MODIFICA END --------------------
END_WHILE
if SysFileEOF(hFile) = 0 
	then Message:='Reading Lux_Psg File: OK';
end_if

//xwDimFile:=SysFileGetSize(sFileName,ADR(hRes));
(* Close file *)
SysFileClose(hFile);

END_FUNCTION_BLOCK

// Utils Functions/OpenFiles_Default_LUX_FB
//Esegue la lettura del file x_DEF_LUX.txt per poi definire come è la configurazione di default dei lux
FUNCTION_BLOCK OpenFiles_Default_LUX_FB
VAR_INPUT
END_VAR
VAR_OUTPUT
	Message		: STRING;
END_VAR
VAR
	hMode		: ACCESS_MODE;
	hFile		: RTS_IEC_HANDLE;
	hRes		: RTS_IEC_RESULT;
	bList		: ARRAY [0..15] OF BYTE;
	i			: DWORD;
	j			: DWORD;
	k			: byte;
	xwDimFile	: LWORD;
	bChar		: BYTE;
	sFileName 	: STRING;
END_VAR

Message:='';
(* Open data file *)
sFileName:=CONCAT(STR1:=MapConf_Path, STR2:=PLC_ID);
sFileName:=CONCAT(STR1:=sFileName, STR2:=DefaultLux_FileName);
hFile:=SysFileOpen(sFileName,AM_READ,ADR(hRes));

(* File not found *)
IF hFile=RTS_INVALID_HANDLE THEN
	Message:='File not found';
	RETURN;
END_IF

(* Close file *)
SysFileClose(hFile);

(* Open data file *)
i:=0;
j:=0;
k:=0;
hFile:=SysFileOpen(sFileName,hMode,ADR(hRes));
//-------------- MODIFICA START --------------------
	SysFileSetPos(hFile, i);	
	SysFileRead(hFile, ADR(bList[j]), 1, ADR(hRes));
//-------------- MODIFICA END --------------------
WHILE SysFileEOF(hFile)<> 0 DO
//-------------- MODIFICA START --------------------	
//	SysFileSetPos(hFile, i);	
//	SysFileRead(hFile, ADR(bList[j]), 1, ADR(hRes));
//-------------- MODIFICA END --------------------	
	IF bList[j] = 16#2F  // se trovo '/'
		THEN 
			SysFileSetPos(hFile, i+1);	
			SysFileRead(hFile, ADR(bList[j+1]), 1, ADR(hRes));
			IF bList[j+1] = 16#2F  // se trovo ancora '/'
				THEN 
					WHILE  bList[j]<> 16#0D DO
						i := i+1;
						SysFileSetPos(hFile, i);	
						SysFileRead(hFile, ADR(bList[j]), 1, ADR(hRes));
					END_WHILE	
					i := i+1;
					SysFileSetPos(hFile, i);	
					SysFileRead(hFile, ADR(bList[j]), 1, ADR(hRes));
					IF bList[j] = 16#0A
						THEN 
							i := i+1;
							j := 0;
							SysFileSetPos(hFile, i);	
							SysFileRead(hFile, ADR(bList[j]), 1, ADR(hRes)); //leggo il primo carattere della nuova riga
						ELSE 
							Message:='Errore 0D 0A';
							RETURN;
					END_IF
				ELSE 
					Message:='Errore //';
					RETURN;
			END_IF
	END_IF
	IF bList[j] <> 16#3B //finchè non trovo ;
		THEN 
			i:=i+1;
			j:=j+1;	
		ELSE
			i:=i+3; //Se trovo ; inizio a salvare i dati della riga letta in TabDefaultLux[k]....
			j:=0;
			k:=k+1;
			TabDefaultLux[k].LuxNumber := ((bList[0]-16#30)*100) + ((bList[1]-16#30)*10) + ((bList[2]-16#30)); //memorizzo il nomero del lux
			TabDefaultLux[k].Mode :=  (bList[4]-16#30)*10 + (bList[5]-16#30); //memorizzo modalità di funzionamento del lux
	END_IF	
//-------------- MODIFICA START --------------------
	SysFileSetPos(hFile, i);	
	SysFileRead(hFile, ADR(bList[j]), 1, ADR(hRes));
//-------------- MODIFICA END --------------------
END_WHILE
if SysFileEOF(hFile) = 0 
	then Message:='Reading Default_Lux File: OK';
end_if

(* Close file *)
SysFileClose(hFile);

END_FUNCTION_BLOCK

// Utils Functions/OpenFiles_CFG_FB
//Esegue la lettura del file CFG.txt all'interno del quale si trovano i dati iniziali di configurazione
FUNCTION_BLOCK OpenFiles_CFG_FB
VAR_INPUT
	//sFileName : STRING;
END_VAR
VAR_OUTPUT
	Message		: STRING;
END_VAR
VAR
	hMode		: ACCESS_MODE;
	hFile		: RTS_IEC_HANDLE;
	hRes		: RTS_IEC_RESULT;
	bList		: ARRAY [0..79] OF BYTE;
	i			: DWORD; //Dim max file: 2^32 byte
	j			: BYTE; //Indice dell'array bList
	x			: BYTE;
	//xwDimFile	: LWORD;
	sFileName, TodString 	: STRING;
	TimerValue				: WORD;
END_VAR

Message:='';
(* Open data file *)
sFileName:=CONCAT(STR1:=MapConf_Path, STR2:=Cfg_FileName);
hFile:=SysFileOpen(sFileName,AM_READ,ADR(hRes));

(* File not found *)
IF hFile=RTS_INVALID_HANDLE THEN
	Message:='File cfg not found';
	RETURN;
END_IF

(* Close file *)
SysFileClose(hFile);

(* Open data file *)
i:=0; //indice di scorrimento del file
j:=0; //indice di scorrimento dell'array dove viene momentaneamente memorizzata la riga prima del ;
hFile:=SysFileOpen(sFileName,hMode,ADR(hRes));
//-------------- MODIFICA START --------------------
	SysFileSetPos(hFile, i);	
	SysFileRead(hFile, ADR(bList[j]), 1, ADR(hRes));
//-------------- MODIFICA END --------------------
WHILE SysFileEOF(hFile)<> 0 DO
//	SysFileSetPos(hFile, i);	
//	SysFileRead(hFile, ADR(bList[j]), 1, ADR(hRes));
	IF bList[j] = 16#2F  // se trovo '/'
		THEN 
			SysFileSetPos(hFile, i+1);	
			SysFileRead(hFile, ADR(bList[j+1]), 1, ADR(hRes));
			IF bList[j+1] = 16#2F  // se trovo ancora '/'
				THEN 
					WHILE  bList[j]<> 16#0D DO
						i := i+1;
						SysFileSetPos(hFile, i);	
						SysFileRead(hFile, ADR(bList[j]), 1, ADR(hRes));
					END_WHILE	
					i := i+1;
					SysFileSetPos(hFile, i);	
					SysFileRead(hFile, ADR(bList[j]), 1, ADR(hRes));
					IF bList[j] = 16#0A
						THEN 
							i := i+1;
							j := 0;
							SysFileSetPos(hFile, i);	
							SysFileRead(hFile, ADR(bList[j]), 1, ADR(hRes)); //leggo il primo carattere della nuova riga
						ELSE 
							Message:='Errore 0D 0A';
							RETURN;
					END_IF
				ELSE 
					Message:='Errore //';
					RETURN;
			END_IF
	END_IF
	IF bList[j] <> 16#3B //finchè non trovo ;
		THEN 
			i:=i+1;
			j:=j+1;	
		ELSE
			i:=i+3; //Se trovo ; inizio a salvare i dati della riga letta in TabLuxPsg[k]....
			j:=0;
			x:=0;
			WHILE (bList[x]<>16#3B) DO  //bList[x]<>';'
				CASE (bList[x]) OF
				(*C*)16#43: TabCfg.id_Clevergy := ((bList[x+1]-16#30)*1000+(bList[x+2]-16#30)*100+(bList[x+3]-16#30)*10+(bList[x+4]-16#30));
				(*P*)16#50: TabCfg.id_Plc := ((bList[x+1]-16#30)*10+(bList[x+2]-16#30));
				(*T*)16#54: 
						(*	TodString := concat(BYTE_TO_STRING(bList[x+1]-16#30),BYTE_TO_STRING(bList[x+2]-16#30));
							TodString := concat(TodString,':');
							TodString := concat(TodString,BYTE_TO_STRING((bList[x+4]-16#30)));
							TodString := concat(TodString,BYTE_TO_STRING((bList[x+5]-16#30)));
							*)							
							TabCfg.HourOfControl := (bList[x+1]-16#30)*10+(bList[x+2]-16#30);	
							TabCfg.MinOfControl := (bList[x+4]-16#30)*10+(bList[x+5]-16#30);

				(*E*)16#45:	TimerValue := ((bList[x+1]-16#30)*1000+(bList[x+2]-16#30)*100+(bList[x+3]-16#30)*10 +(bList[x+4]-16#30));
							TabCfg.TimeOutError := DWORD_TO_TIME(TimerValue*1000); 
				END_CASE
				x:=x+1;
			END_WHILE
	END_IF	
//-------------- MODIFICA START --------------------
	SysFileSetPos(hFile, i);	
	SysFileRead(hFile, ADR(bList[j]), 1, ADR(hRes));
//-------------- MODIFICA END --------------------
END_WHILE
if SysFileEOF(hFile) = 0 
	then
		Message:='Reading Cfg File: OK';
		Plant_SN := word_to_dword(TabCfg.id_Clevergy);    
		PLC_ID := byte_to_string(TabCfg.id_Plc);
		Plant_NAME:=REPLACE(Plant_NAME,word_to_string(TabCfg.id_Clevergy),2,6);
		
end_if

//xwDimFile:=SysFileGetSize(sFileName,ADR(hRes));
(* Close file *)
SysFileClose(hFile);

END_FUNCTION_BLOCK

// Utils Functions/FileCopyToSD_FB
FUNCTION_BLOCK FileCopyToSD_FB
VAR_INPUT
END_VAR
VAR_OUTPUT
	Message		: STRING;
END_VAR
VAR
	hMode		: ACCESS_MODE;
	hFile		: RTS_IEC_HANDLE;
	hRes		: RTS_IEC_RESULT;
	DestFile	: STRING;
	SourceFile	: STRING;
	DestDir		: STRING;
	xwDimFile	: LWORD;
	ptDim		: POINTER TO LWORD;
	FileCopying	: BOOL;
END_VAR

FileCopying := FALSE;

//SourceFile := '1_DEF_LUX.txt';
//DestFile := '/media/sd/1_DEF_LUX_copy.txt';
DestDir := '/media/sd/';
DestFile := CONCAT(STR1:=DestDir, STR2:=SourceFile);
hFile:=SysFileOpen(DestFile,AM_READ,ADR(hRes));
(*
IF hFile<>RTS_INVALID_HANDLE THEN //Se il file è già presente
	Message:='File found';
	//implementare il messaggio che il file sarà sovrascritto
	SysFileClose(hFile);
	RETURN;
END_IF
*)

xwDimFile:=SysFileGetSize(SourceFile,ADR(hRes));
ptDim:= ADR(xwDimFile);
hRes:=SysFileCopy(DestFile, SourceFile,ptDim);
IF hRes = 0 
	THEN
		Message:='Copia su SD eseguita';	
		FileCopying := TRUE;
END_IF

END_FUNCTION_BLOCK

// Utils Functions/FileCopySDToPLC_FB
FUNCTION_BLOCK FileCopySDToPLC_FB
VAR_INPUT
END_VAR
VAR_OUTPUT
	Message		: STRING;
END_VAR
VAR
	hMode		: ACCESS_MODE;
	hFile		: RTS_IEC_HANDLE;
	hRes		: RTS_IEC_RESULT;
	DestFile	: STRING;
	SourceFile, SourceFileOnSD	: STRING;
	DestDir, SourceDir		: STRING;
	xwDimFile	: LWORD;
	ptDim		: POINTER TO LWORD;
	FileCopying	: BOOL;
END_VAR

FileCopying := FALSE;

//SourceFile := '1_DEF_LUX.txt';
//DestFile := '/media/sd/1_DEF_LUX_copy.txt';
DestFile:=SourceFile;	
SourceDir := '/media/sd/';
SourceFile := CONCAT(STR1:=SourceDir, STR2:=SourceFile);
(*
hFile:=SysFileOpen(DestFile,AM_READ,ADR(hRes));

IF hFile<>RTS_INVALID_HANDLE THEN //Se il file è già presente
	Message:='File found';
	//implementare il messaggio che il file sarà sovrascritto
	SysFileClose(hFile);
	RETURN;
END_IF
*)

xwDimFile:=SysFileGetSize(SourceFile,ADR(hRes));
ptDim:= ADR(xwDimFile);
hRes:=SysFileCopy(DestFile, SourceFile,ptDim);
IF hRes = 0 
	THEN
		Message:='Copia su PLC eseguita';	
		FileCopying := TRUE;
END_IF

END_FUNCTION_BLOCK

// Utils Functions/FileSize_and_Time_FB
FUNCTION_BLOCK FileSize_and_Time_FB
VAR_INPUT
END_VAR
VAR_OUTPUT
	Message		: STRING;
	MessageBK		: STRING;
END_VAR
VAR
	hMode		: ACCESS_MODE;
	hFile		: RTS_IEC_HANDLE;
	hRes		: RTS_IEC_RESULT;
	FileTime	: SYS_FILETIME;
	DestFile	: STRING;
	SourceFile	: STRING;
	DestDir		: STRING;
	xwDimFile	: LWORD;
	ptDim		: POINTER TO LWORD;
	xwDimFileBK	: LWORD;
	ptDimBK		: POINTER TO LWORD;
	FileCopying	: BOOL;
	LastModifyT	: DT;
	LastModifyS	: STRING;
	LastModifyTBK	: DT;
	LastModifySBK	: STRING;
	
END_VAR

FileCopying := FALSE;

//SourceFile := '1_DEF_LUX.txt';
//DestFile := '/media/sd/1_DEF_LUX_copy.txt';
DestDir := '/media/sd/';
SourceFile := 'LOG.DAT';
DestFile := CONCAT(STR1:=DestDir, STR2:=SourceFile);
hFile:=SysFileOpen(DestFile,AM_READ,ADR(hRes));
(*
IF hFile<>RTS_INVALID_HANDLE THEN //Se il file è già presente
	Message:='File found';
	//implementare il messaggio che il file sarà sovrascritto
	SysFileClose(hFile);
	RETURN;
END_IF
*)
hRes:=SysFileGetTime(DestFile,ADR(FileTime));
if  hRes = 0
	then
		LastModifyT:= udint_to_dt(FileTime.tLastModification);
		LastModifyS:= dt_to_string(LastModifyT);
	//
end_if
xwDimFile:=SysFileGetSize(DestFile,ADR(hRes));
Message := lword_to_string(xwDimFile);
ptDim:= ADR(xwDimFile);

DestDir := '/media/sd/';
SourceFile := 'LOG.BCK';
DestFile := CONCAT(STR1:=DestDir, STR2:=SourceFile);
hFile:=SysFileOpen(DestFile,AM_READ,ADR(hRes));

hRes:=SysFileGetTime(DestFile,ADR(FileTime));
if  hRes = 0
	then
		LastModifyTBK:= udint_to_dt(FileTime.tLastModification);
		LastModifySBK:= dt_to_string(LastModifyTBK);
	//
end_if
xwDimFileBK:=SysFileGetSize(DestFile,ADR(hRes));
MessageBK := lword_to_string(xwDimFileBK);
ptDimBK:= ADR(xwDimFileBK);

(*
hRes:=SysFileCopy(DestFile, SourceFile,ptDim);
IF hRes = 0 
	THEN
		Message:='Copia su SD eseguita';	
		FileCopying := TRUE;
END_IF*)

END_FUNCTION_BLOCK

// Utils Functions/LuxTimerModify_FB
FUNCTION_BLOCK LuxTimerModify_FB
VAR_INPUT
	NewValueTimer: dword;
	IdFind:	word;
END_VAR
VAR_OUTPUT
END_VAR
VAR
	x		: word;
	counter	: word;
END_VAR

x:=1;
while (IdFind <> TabLuxPsg[x].LuxId) and ( x <= MAX_LUXNUM) do
x := x + 1;	
END_WHILE
if IdFind = TabLuxPsg[x].LuxId 
	then TabLuxPsg[x].TimerOn := dword_to_time(NewValueTimer*1000);
	for counter := 1 to MAX_LUXNUM do
		if LuxElement[counter].ID = IdFind
			then LuxElement[counter].LuxTimer := dword_to_time(NewValueTimer*1000); // TabLuxPsg[x].TimerOn; //set del nuovo valore del timer del lux 	
		end_if
	END_FOR
END_IF

END_FUNCTION_BLOCK

// Utils Functions/LuxManOnOff_FB
FUNCTION_BLOCK LuxManOnOff_FB
VAR_INPUT
	NewValueManSw0: byte;
	NewValueManSw1: byte;
	IdFind:	word;
END_VAR
VAR_OUTPUT
END_VAR
VAR
	NewValueManOnOff: byte;
	x,	counter		: word;
END_VAR

x:=1;
NewValueManOnOff := NewValueManSw1 * 2 + NewValueManSw0 * 1;
if NewValueManOnOff = 3 
	then NewValueManOnOff := 2; //blocco la commutazione al mode 03 che è riservata ai timer con on su passaggio
end_if
counter:=0;
while (IdFind <> TabDefaultLux[x].LuxNumber) and ( x <= MAX_LUXNUM) do
x := x + 1;	
end_while
if IdFind = TabDefaultLux[x].LuxNumber 
	then 
	if TabDefaultLux[x].Mode <> 3 
		then
			TabDefaultLux[x].Mode := NewValueManOnOff;
			while (LuxElement[counter].ID <> IdFind) and ( counter <= MAX_LUXNUM) do
				counter := counter + 1;
			end_while
			if IdFind = LuxElement[counter].ID
				then LuxElement[counter].CTRL_MODE := NewValueManOnOff;	//TabDefaultLux[x].Mode; //copio il mode nella tabella delle variabili dei lux
			end_if
		end_if
end_if

END_FUNCTION_BLOCK

// Utils/RTC_Update
FUNCTION RTC_Update : BOOL
VAR
	T: DT;
	TS: STRING;
	TS2: STRING;
	Hour: BYTE;
	Minute: BYTE;
END_VAR

(* Get RTC time *)
T:=SysRtcGetTime(TRUE);
Sys.Time_CT_DT:=T;
(* Calculate variables *)
TS:=DT_TO_STRING(T);
Sys.Time_LogString:=DELETE(STR:=TS, LEN:=3, POS:=1);
TS2:=MID(STR:=TS, LEN:=4, POS:= 4); 
Sys.Time_Year 	:=STRING_TO_WORD(TS2);
TS2:=MID(STR:=TS, LEN:=2, POS:= 9); 
Sys.Time_Month	:=STRING_TO_BYTE(TS2);
TS2:=MID(STR:=TS, LEN:=2, POS:=12); 
Sys.Time_Day  	:=STRING_TO_BYTE(TS2);
Sys.Time_CT_Day:=(32*(Sys.Time_Month-1)+Sys.Time_Day-1);
TS2:=MID(STR:=TS, LEN:=2, POS:=15); 
Hour			:=STRING_TO_BYTE(TS2);
Sys.Time_Hour := Hour;
TS2:=MID(STR:=TS, LEN:=2, POS:=18); 
Minute		 	:=STRING_TO_BYTE(TS2);
Sys.Time_Min := Minute;
Sys.Time_CT_Quarter:=Hour*4+(Minute/15);

END_FUNCTION

// Utils/CSV_Log
FUNCTION CSV_Log : BOOL
VAR_INPUT
END_VAR
VAR CONSTANT
	LogFileName:STRING:='S:\LOGS_ID4V3.CSV';
END_VAR
VAR
	s1 : STRING(256);
	hFile: 	DWORD;
END_VAR

(* Check file presence *)
hFile:=SysFileOpen(LogFileName,'r');
IF hFile=0 THEN
	(*** File not exist *** Create file and write header *)
	hFile:=SysFileOpen(LogFileName,'w');
	IF hFile<>0 THEN
		(* Write CSV header *)
		s1:='Title1;Title2,...';
		SysFileWrite(hFile, ADR(s1), LEN(s1));
		SysFileWrite(hFile, ADR(Logger_CRLF), LEN(Logger_CRLF));
	END_IF
ELSE
	(*** File exist *** Close file and reopen in append mode *)
	SysFileClose(hFile);
	hFile:=SysFileOpen(LogFileName,'a');
END_IF

(* Log to file *)
IF hFile<>0 THEN
	(* Date stamp *)
	s1:=REPLACE( Sys.Time_LogString , ' ' , 1 , 11 );
	SysFileWrite(hFile, ADR(s1), LEN(s1));
	(* Write CSV data *)
	s1:=CONCAT(';', 'Data1' );
	s1:=CONCAT(s1 , ';');
	s1:=CONCAT(s1 , 'Data2' );
	s1:=CONCAT(s1 , ';');
	s1:=CONCAT(s1 , '...' );
	SysFileWrite(hFile, ADR(s1), LEN(s1));
	(* Add line CRLF and close *)
	SysFileWrite(hFile, ADR(Logger_CRLF), LEN(Logger_CRLF));
	SysFileClose(hFile);
END_IF

END_FUNCTION

// PLC_RT
PROGRAM PLC_RT
VAR
	x, y, k	: BYTE;
END_VAR

(******************************************************************************
 ****                       HP TASK CODE	                               ****
 ******************************************************************************
*)

(*==============================*)
(*== Running cycle operations ==*)
(*==============================*)
//IF SYS.Status>S_INIT_VAR THEN
IF TRUE THEN
	(* Execute cycle processes *)
	AsiInMapping();
	AsiOutMapping();
	k := 1;
	FOR x:= 1 TO ASI_TOT DO
		CASE TabAsiPsg[x].Asi1_2 OF
			1: FOR y := 0 TO MAX_BIT DO
					IF TabAsiPsg[x].bit_psg[y] <> 0
					THEN //eseguo operazione indicizzata come la seguente: PSG[89](Psg_state:=ASI_1[ASI_A, 1,0], NumTransition:=PsgCounter[89]);
						PSG[k].ID := TabAsiPsg[x].bit_psg[y];
						PSG[k](Psg_state:=ASI_1[TabAsiPsg[x].A_B, TabAsiPsg[x].Address, y], NumTransition:=PsgCounter[k]);
						k:=k+1;
						  
					END_IF
				END_FOR
			2: FOR y := 0 TO MAX_BIT DO
					IF TabAsiPsg[x].bit_psg[y] <> 0
					THEN //eseguo operazione indicizzata come la seguente: PSG[29](Psg_state:=ASI_2[ASI_A, 1,0], NumTransition:=PsgCounter[29]);
						PSG[k].ID := TabAsiPsg[x].bit_psg[y];
						PSG[k](Psg_state:=ASI_2[TabAsiPsg[x].A_B, TabAsiPsg[x].Address, y], NumTransition:=PsgCounter[k]);
						k:=k+1;						
					END_IF
				END_FOR
		END_CASE
	END_FOR;	
END_IF

END_PROGRAM

// Utils Functions/AsiInMapping
FUNCTION AsiInMapping : BOOL
VAR_INPUT
END_VAR
VAR
	x, y: BYTE;
END_VAR

FOR x:= 1 TO ASI_TOT DO
	CASE TabAsiPsg[x].Asi1_2 OF
		1: FOR y := 0 TO MAX_BIT DO
				IF TabAsiPsg[x].bit_psg[y] <> 0
				THEN
					ASI_1[TabAsiPsg[x].A_B, TabAsiPsg[x].Address, y] := PSG_LIST[TabAsiPsg[x].bit_psg[y]];
				END_IF
			END_FOR
		2: FOR y := 0 TO MAX_BIT DO
				IF TabAsiPsg[x].bit_psg[y] <> 0
				THEN
					ASI_2[TabAsiPsg[x].A_B, TabAsiPsg[x].Address, y] := PSG_LIST[TabAsiPsg[x].bit_psg[y]];
				END_IF
			END_FOR
	END_CASE
END_FOR;	
(*
FOR y:= 1 TO LUXM_MAX DO //1...900
		LUX_LIST[y] := LuxOutput_ASI[y];
END_FOR;	
*)
(*
//----------------------------- Start - Mapping ingressi ASI 1 A ----------------------------- 
//ASI_1_A[1,0]:=PSG_LIST[89];	//PSG89_IN;
//ASI_1_A[1,2]:=PSG_LIST[90];	//PSG90_IN;
ASI_1_A[2,0]:=PSG_LIST[91];	//PSG91_IN;
ASI_1_A[2,2]:=PSG_LIST[92];	//PSG92_IN;
ASI_1_A[3,0]:=PSG93_IN;
ASI_1_A[3,2]:=PSG94_IN;
ASI_1_A[4,0]:=PSG95_IN;
ASI_1_A[4,2]:=PSG96_IN;
ASI_1_A[5,0]:=PSG97_IN;
ASI_1_A[5,2]:=PSG98_IN;
ASI_1_A[6,0]:=PSG99_IN;
ASI_1_A[6,2]:=PSG100_IN;
ASI_1_A[7,0]:=PSG101_IN;
ASI_1_A[7,2]:=PSG102_IN;
ASI_1_A[8,0]:=PSG103_IN;
ASI_1_A[8,2]:=PSG104_IN;
ASI_1_A[9,0]:=PSG105_IN;
ASI_1_A[9,2]:=PSG106_IN;
ASI_1_A[10,0]:=PSG107_IN;
ASI_1_A[10,2]:=PSG108_IN;
ASI_1_A[11,0]:=PSG109_IN;
ASI_1_A[11,2]:=PSG110_IN;
ASI_1_A[12,0]:=PSG111_IN;
ASI_1_A[12,2]:=PSG112_IN;
ASI_1_A[13,0]:=PSG113_IN;
ASI_1_A[13,2]:=PSG114_IN;
ASI_1_A[14,0]:=PSG115_IN;
ASI_1_A[14,2]:=PSG116_IN;
ASI_1_A[15,0]:=PSG117_IN;
ASI_1_A[15,2]:=PSG118_IN;
ASI_1_A[16,0]:=PSG119_IN;
ASI_1_A[16,2]:=PSG120_IN;
 
ASI_1_A[17,0]:=PSG149_IN;
ASI_1_A[17,2]:=PSG150_IN;
ASI_1_A[18,0]:=PSG151_IN;
ASI_1_A[18,2]:=PSG152_IN;
ASI_1_A[19,0]:=PSG153_IN;
ASI_1_A[19,2]:=PSG154_IN;
ASI_1_A[20,0]:=PSG155_IN;
ASI_1_A[20,2]:=PSG156_IN;
ASI_1_A[21,0]:=PSG157_IN;
ASI_1_A[21,2]:=PSG158_IN;
ASI_1_A[22,0]:=PSG159_IN;
ASI_1_A[22,2]:=PSG160_IN;
ASI_1_A[23,0]:=PSG161_IN;
ASI_1_A[23,2]:=PSG162_IN;
ASI_1_A[24,0]:=PSG163_IN;
ASI_1_A[24,2]:=PSG164_IN;
ASI_1_A[25,0]:=PSG165_IN;
ASI_1_A[25,2]:=PSG166_IN;
ASI_1_A[26,0]:=PSG167_IN;
ASI_1_A[26,2]:=PSG168_IN;
ASI_1_A[27,0]:=PSG169_IN;
ASI_1_A[27,2]:=PSG170_IN;
ASI_1_A[28,0]:=PSG171_IN;
ASI_1_A[28,2]:=PSG172_IN;
ASI_1_A[29,0]:=PSG173_IN;
ASI_1_A[29,2]:=PSG174_IN;
ASI_1_A[30,0]:=PSG175_IN;
ASI_1_A[30,2]:=PSG176_IN;
ASI_1_A[31,0]:=PSG177_IN;
ASI_1_A[31,2]:=PSG178_IN;
//----------------------------- End - Mapping ingressi ASI 1 A -----------------------------
//----------------------------- Start - Mapping ingressi ASI 1 B ----------------------------
ASI_1_B[1,0]:=PSG179_IN;
ASI_1_B[1,2]:=PSG180_IN;
ASI_1_B[2,0]:=LUXST_46;
ASI_1_B[3,0]:=LUXST_47;
ASI_1_B[4,0]:=LUXST_48;


//----------------------------- Start - Mapping ingressi ASI 2 A ----------------------------
ASI_2_A[1,0]:=PSG29_IN;
ASI_2_A[1,2]:=PSG30_IN;
ASI_2_A[2,0]:=PSG31_IN;
ASI_2_A[2,2]:=PSG32_IN;
ASI_2_A[3,0]:=PSG33_IN;
ASI_2_A[3,2]:=PSG34_IN;
ASI_2_A[4,0]:=PSG35_IN;
ASI_2_A[4,2]:=PSG36_IN;
ASI_2_A[5,0]:=PSG37_IN;
ASI_2_A[5,2]:=PSG38_IN;
ASI_2_A[6,0]:=PSG39_IN;
ASI_2_A[6,2]:=PSG40_IN;
ASI_2_A[7,0]:=PSG41_IN;
ASI_2_A[7,2]:=PSG42_IN;
ASI_2_A[8,0]:=PSG43_IN;
ASI_2_A[8,2]:=PSG44_IN;
ASI_2_A[9,0]:=PSG45_IN;
ASI_2_A[9,2]:=PSG46_IN;
ASI_2_A[10,0]:=PSG47_IN;
ASI_2_A[10,2]:=PSG48_IN;
ASI_2_A[11,0]:=PSG49_IN;
ASI_2_A[11,2]:=PSG50_IN;
ASI_2_A[12,0]:=PSG51_IN;
ASI_2_A[12,2]:=PSG52_IN;
ASI_2_A[13,0]:=PSG53_IN;
ASI_2_A[13,2]:=PSG54_IN;
ASI_2_A[14,0]:=PSG55_IN;
ASI_2_A[14,2]:=PSG56_IN;
ASI_2_A[15,0]:=PSG57_IN;
ASI_2_A[15,2]:=PSG58_IN;
ASI_2_A[16,0]:=PSG59_IN;
ASI_2_A[16,2]:=PSG60_IN;

ASI_2_A[17,0]:=PSG209_IN;
ASI_2_A[17,2]:=PSG210_IN;
ASI_2_A[18,0]:=PSG211_IN;
ASI_2_A[18,2]:=PSG212_IN;
ASI_2_A[19,0]:=PSG213_IN;
ASI_2_A[19,2]:=PSG214_IN;
ASI_2_A[20,0]:=PSG215_IN;
ASI_2_A[20,2]:=PSG216_IN;
ASI_2_A[21,0]:=PSG217_IN;
ASI_2_A[21,2]:=PSG218_IN;
ASI_2_A[22,0]:=PSG219_IN;
ASI_2_A[22,2]:=PSG220_IN;
ASI_2_A[23,0]:=PSG221_IN;
ASI_2_A[23,2]:=PSG222_IN;
ASI_2_A[24,0]:=PSG223_IN;
ASI_2_A[24,2]:=PSG224_IN;
ASI_2_A[25,0]:=PSG225_IN;
ASI_2_A[25,2]:=PSG226_IN;
ASI_2_A[26,0]:=PSG227_IN;
ASI_2_A[26,2]:=PSG228_IN;
ASI_2_A[27,0]:=PSG229_IN;
ASI_2_A[27,2]:=PSG230_IN;
ASI_2_A[28,0]:=PSG231_IN;
ASI_2_A[28,2]:=PSG232_IN;
ASI_2_A[29,0]:=PSG233_IN;
ASI_2_A[29,2]:=PSG234_IN;
ASI_2_A[30,0]:=PSG235_IN;
ASI_2_A[30,2]:=PSG236_IN;
ASI_2_A[31,0]:=PSG237_IN;
ASI_2_A[31,2]:=PSG238_IN;
//----------------------------- End - Mapping ingressi ASI 2 A -----------------------------
//----------------------------- Start - Mapping ingressi ASI 2 B -----------------------------
ASI_2_B[1,0]:=PSG239_IN;
ASI_2_B[1,2]:=PSG240_IN;

ASI_2_B[2,0]:=LUXST_07;
ASI_2_B[2,2]:=LUXST_08;
ASI_2_B[3,0]:=LUXST_09;
ASI_2_B[3,2]:=LUXST_10;
ASI_2_B[4,0]:=LUXST_11;
ASI_2_B[4,2]:=LUXST_12;
ASI_2_B[5,0]:=LUXST_27;
ASI_2_B[5,2]:=LUXST_28;
ASI_2_B[6,0]:=LUXST_29;
ASI_2_B[6,2]:=LUXST_30;
ASI_2_B[7,0]:=LUXST_31;
ASI_2_B[7,2]:=LUXST_32;
ASI_2_B[8,0]:=LUXST_33;
ASI_2_B[8,2]:=LUXST_34;
ASI_2_B[9,0]:=LUXST_35;
ASI_2_B[9,2]:=LUXST_36;
ASI_2_B[10,0]:=LUXST_37;
ASI_2_B[10,2]:=LUXST_38;
ASI_2_B[11,0]:=LUXST_39;
ASI_2_B[11,2]:=LUXST_40;
ASI_2_B[12,0]:=LUXST_41;
ASI_2_B[12,2]:=LUXST_42;
ASI_2_B[13,0]:=LUXST_105;
ASI_2_B[13,1]:=LUXST_106;
ASI_2_B[13,2]:=LUXST_107;
ASI_2_B[13,3]:=LUXST_108;
ASI_2_B[14,0]:=LUXST_109;
ASI_2_B[14,1]:=LUXST_110;
ASI_2_B[14,2]:=LUXST_111;
ASI_2_B[14,3]:=LUXST_112;
ASI_2_B[15,0]:=LUXST_113;
ASI_2_B[15,1]:=LUXST_114;
ASI_2_B[15,2]:=LUXST_115;
ASI_2_B[15,3]:=LUXST_116;
ASI_2_B[16,0]:=LUXST_117;
ASI_2_B[16,1]:=LUXST_118;
ASI_2_B[16,2]:=LUXST_119;
ASI_2_B[16,3]:=LUXST_120;
ASI_2_B[17,0]:=LUXST_121;
ASI_2_B[17,1]:=LUXST_122;
ASI_2_B[17,2]:=LUXST_123;
ASI_2_B[17,3]:=LUXST_124;
ASI_2_B[18,0]:=LUXST_125;
ASI_2_B[18,1]:=LUXST_126;
ASI_2_B[18,2]:=LUXST_127;
ASI_2_B[18,3]:=LUXST_128;
ASI_2_B[19,0]:=LUXST_129;
ASI_2_B[19,1]:=LUXST_130;
ASI_2_B[19,2]:=LUXST_131;
ASI_2_B[19,3]:=LUXST_132;
ASI_2_B[20,0]:=LUXST_133;
ASI_2_B[20,1]:=LUXST_134;
ASI_2_B[20,2]:=LUXST_135;
ASI_2_B[20,3]:=LUXST_136;
ASI_2_B[21,0]:=LUXST_137;
ASI_2_B[21,1]:=LUXST_138;
ASI_2_B[21,2]:=LUXST_139;
ASI_2_B[21,3]:=LUXST_140;
ASI_2_B[22,0]:=LUXST_141;
ASI_2_B[22,1]:=LUXST_142;
ASI_2_B[22,2]:=LUXST_143;
ASI_2_B[22,3]:=LUXST_144;
ASI_2_B[23,0]:=LUXST_145;
ASI_2_B[23,1]:=LUXST_146;
ASI_2_B[23,2]:=LUXST_147;
ASI_2_B[23,3]:=LUXST_148;
ASI_2_B[24,0]:=LUXST_149;
ASI_2_B[24,1]:=LUXST_150;
ASI_2_B[24,2]:=LUXST_151;
ASI_2_B[24,3]:=LUXST_152;
ASI_2_B[25,0]:=LUXST_153;
ASI_2_B[25,1]:=LUXST_154;
ASI_2_B[25,2]:=LUXST_155;
ASI_2_B[25,3]:=LUXST_156;
ASI_2_B[26,0]:=LUXST_157;
ASI_2_B[26,1]:=LUXST_158;
ASI_2_B[26,2]:=LUXST_159;
ASI_2_B[26,3]:=LUXST_160;
ASI_2_B[27,0]:=LUXST_161;
ASI_2_B[27,1]:=LUXST_162;
ASI_2_B[27,2]:=LUXST_163;
ASI_2_B[27,3]:=LUXST_164;
ASI_2_B[28,0]:=LUXST_165;
ASI_2_B[28,1]:=LUXST_166;
ASI_2_B[28,2]:=LUXST_167;
ASI_2_B[28,3]:=LUXST_168;
//----------------------------- End - Mapping ingressi ASI 2 B -----------------------------
*)

END_FUNCTION

// Utils Functions/AsiOutMapping
FUNCTION AsiOutMapping : BOOL
VAR_INPUT
END_VAR
VAR
	x: BYTE;
	y: WORD;
END_VAR

//----------------------------- Start - Mapping uscite ASI 1 A ----------------------------- 
(*
FOR x:= 1 TO ASI_TOT DO
	CASE TabASILux[x].Asi1_2 OF
		1: FOR y := 0 TO MAX_BIT DO
				IF TabASILux[x].bit_lux[y] <> 0
				THEN //eseguo il mapping delle uscite lux ponendo a 1 quelle attive  e rilevate dai files di configurazione
					 // es. LUX_LIST[105] := 1 perchè il lux con id 105 è presente nel listato
					LUX_LIST[TabASILux[x].bit_lux[y]] := ASI_1[TabASILux[x].A_B, TabASILux[x].Address, y];
				END_IF
			END_FOR
		2: FOR y := 0 TO MAX_BIT DO
				IF TabASILux[x].bit_lux[y] <> 0
				THEN //come sopra per asi 2
					LUX_LIST[TabASILux[x].bit_lux[y]] := ASI_2[TabASILux[x].A_B, TabASILux[x].Address, y];
				END_IF
			END_FOR
	END_CASE
END_FOR *)
(*
FOR x:= 1 TO ASI_TOT DO
	CASE TabASILux[x].Asi1_2 OF
		1: FOR y := 0 TO MAX_BIT DO
				IF TabASILux[x].bit_lux[y] <> 0
				THEN //eseguo il mapping degli stati dei relè - Per ogni relè in out (lux) corrisponde un bit in input che ne
					//identifica lo stato. Questo pin si trova allo stesso indirizzo dell'uscita del relè, ma ha ovviamento
					//indirizzo di input(Q1.2 ---> I1.2)
					//Lo stato dei relè (input) viene letto della lista LUX_ST[] e va a settare il corrispondente bit della mappa 
					//degli indirizzi asi in ASI_1. Lo stato di questi indirizzi viene usato per acendere di verde lo stato delle luci
					ASI_1[TabASILux[x].A_B, TabASILux[x].Address, y] := LUX_ST[TabASILux[x].bit_lux[y]];
				END_IF
			END_FOR
		2: FOR y := 0 TO MAX_BIT DO
				IF TabASILux[x].bit_lux[y] <> 0
				THEN //come sopra per asi2
					ASI_2[TabASILux[x].A_B, TabASILux[x].Address, y] := LUX_ST[TabASILux[x].bit_lux[y]];
				END_IF
			END_FOR
	END_CASE
END_FOR
*)
	//Aziono lo stato delle uscite sulla base dei valori contenuti in LuxOutput_ASI[y] settati nei rispettivi LuxElement
FOR y:= 1 TO LUXM_MAX_ID DO //1...900
		LUX_LIST[y] := LuxOutput_ASI[y];
END_FOR;	

(*
FOR x:= 1 TO ASI_TOT DO
	CASE TabASILux[x].Asi1_2 OF
		1:	LUX_LIST[TabASILux[x].LUX] := ASI_1[TabASILux[x].A_B, TabASILux[x].Address, TabASILux[x].Bit_address];
		2:	LUX_LIST[TabASILux[x].LUX] := ASI_2[TabASILux[x].A_B, TabASILux[x].Address, TabASILux[x].Bit_address];
	END_CASE	
END_FOR;	
FOR x:= 1 TO ASI_TOT DO
	CASE TabASILux[x].Asi1_2 OF
		1:	ASI_1[TabASILux[x].A_B, TabASILux[x].Address, TabASILux[x].Bit_address] := LUX_ST[TabASILux[x].LUX];
		2: 	ASI_2[TabASILux[x].A_B, TabASILux[x].Address, TabASILux[x].Bit_address] := LUX_ST[TabASILux[x].LUX];
	END_CASE	
END_FOR;	
*)

//----------------------------- End - Mapping uscite ASI 1 A -----------------------------
//----------------------------- Start - Mapping uscite ASI 1 B ----------------------------
//LUX_LIST[46] := LuxOutput_ASI[46];	//ASI_OUT_1_B[2,0];
//,LUXM_47,LUXM_48
//----------------------------- End - Mapping uscite ASI 1 B -----------------------------

//----------------------------- Start - Mapping ingressi ASI 2 A ----------------------------
//ASI_2_A[1,0]:=PSG29_IN;
//----------------------------- End - Mapping ingressi ASI 2 A -----------------------------
//----------------------------- Start - Mapping ingressi ASI 2 B -----------------------------
//ASI_2_B[1,0]:=PSG239_IN;
//----------------------------- End - Mapping ingressi ASI 2 B -----------------------------

END_FUNCTION

// Utils Functions/AVERAGE_DINT
FUNCTION_BLOCK AVERAGE_DINT
VAR_INPUT
	IN: 	DINT;
END_VAR
VAR_OUTPUT
	HI:		DINT;
	AVG:	DINT;
	LOW:	DINT;
	ERR:	BOOL;
END_VAR
VAR
	sum:	REAL;
	cnt:	WORD;
END_VAR

IF cnt>=65000 THEN
	ERR:=TRUE;
	Read();
	sum := sum - DINT_TO_REAL(AVG);
	cnt := cnt - 1;
END_IF

sum := sum + DINT_TO_REAL(IN);
cnt := cnt + 1;

IF IN<LOW THEN LOW:=IN; END_IF
IF IN>HI  THEN HI :=IN; END_IF

ACTION Read:
AVG := REAL_TO_DINT(sum/cnt);
END_ACTION

ACTION Reset:
HI:=IN;
AVG:=IN;
LOW:=IN;
ERR:=FALSE;

sum:=DINT_TO_REAL(IN);
cnt:=1;
END_ACTION

END_FUNCTION_BLOCK

// Utils Functions/AVERAGE_T
FUNCTION_BLOCK AVERAGE_T
VAR_INPUT
	IN: 	INT;
END_VAR
VAR_OUTPUT
	HI:		INT;
	AVG:	INT;
	LOW:	INT;
	ERR:	BOOL;
END_VAR
VAR
	sum:	DINT;
	cnt:	WORD;
END_VAR

IF cnt>=65000 THEN
	ERR:=TRUE;
	Read();
	sum := sum - AVG;
	cnt := cnt + 1;
END_IF

sum := sum + IN;
cnt := cnt + 1;

IF IN<LOW THEN  LOW:=IN; END_IF
IF IN>HI  THEN HI :=IN; END_IF

ACTION Read:
AVG := DINT_TO_INT(sum/cnt);
END_ACTION

ACTION Reset:
HI:=IN;
AVG:=IN;
LOW:=IN;
ERR:=FALSE;

sum:=IN;
cnt:=1;
END_ACTION

END_FUNCTION_BLOCK

// Utils Functions/COPY_32SWAP16
FUNCTION COPY_32SWAP16:BOOL
VAR_INPUT
	pSourceAddress		:POINTER TO ARRAY[1..2] OF WORD;
	pDestinationAddress	:POINTER TO ARRAY[1..2] OF WORD;
END_VAR
VAR
END_VAR

pDestinationAddress^[1]:=pSourceAddress^[2];
pDestinationAddress^[2]:=pSourceAddress^[1];

END_FUNCTION

// Utils Functions/FLT_TAP
FUNCTION_BLOCK FLT_TAP
VAR_INPUT
	IN		: BOOL;
	TAP		: BYTE:=4;
	INITEV	: BOOL:=TRUE;
END_VAR
VAR_OUTPUT
	OUT		: BOOL;
	EVH		: BOOL;
	EVL		: BOOL;
END_VAR
VAR
	init	: BOOL:=FALSE;
	cnt		: BYTE;
END_VAR

EVH:=FALSE;
EVL:=FALSE;

IF NOT init THEN
	init := TRUE;
	IF INITEV THEN
		OUT  := NOT IN;
		cnt  := TAP;
	ELSE
		OUT  := IN;
	END_IF
END_IF

IF OUT<>IN THEN
	cnt:=cnt+1;
	IF cnt>TAP THEN
		OUT:=IN;
		cnt:=0;
		IF OUT THEN EVH:=TRUE; ELSE EVL:=TRUE; END_IF
	END_IF
ELSE
	cnt:=0;
END_IF

END_FUNCTION_BLOCK

// Utils Functions/LINEAR
FUNCTION LINEAR : REAL (* Linear interpolation *)
VAR_INPUT
	X_In	: REAL;
	P1_X	: REAL;
	P1_Y	: REAL;
	P2_X	: REAL;
	P2_Y	: REAL;
END_VAR
VAR
END_VAR

LINEAR:=P1_Y+(((P2_Y-P1_Y)*(X_In-P1_X))/(P2_X-P1_X));

END_FUNCTION

// Utils Functions/LINEAR_BAD
FUNCTION LINEAR_BAD : INT (* Linear interpolation *)
VAR_INPUT
	PuntoMinX	: INT;
	PuntoMaxX	: INT;
	ValIn		: INT;
	PuntoMinY	: REAL;
	PuntoMaxY	: REAL;
	Decimali	: BYTE;
END_VAR
VAR
	Gain				: REAL;
	PuntoMinX_R			: REAL;
	PuntoMaxX_R			: REAL;
	Linearizzazione_R	: REAL;
END_VAR


PuntoMinX_R:=INT_TO_REAL(PuntoMinX);
PuntoMaxX_R:=INT_TO_REAL(PuntoMaxX);

Gain:=(PuntoMaxX_R-PuntoMinX_R)/(PuntoMaxY-PuntoMinY);	(* Calcolo in guadagno per la linarizzazione *)
Linearizzazione_R:=PuntoMinx+(Gain*(ValIn-PuntoMinY));	(* Ottengo il valore linearizzato *)

LINEAR_BAD:=REAL_TO_INT(Linearizzazione_R*(EXPT(10, Decimali)));  (* Ottengo intero con i decimai voluti *)

END_FUNCTION

// Utils Functions/MEMCLR
FUNCTION MEMCLR:BOOL
VAR_INPUT
	pDestinationAddress:POINTER TO ARRAY[1..2] OF BYTE;
	BytesToClear:WORD;
END_VAR
VAR
END_VAR

WHILE (BytesToClear > 0) DO
	pDestinationAddress^[1]:=0;
	pDestinationAddress:=ADR(pDestinationAddress^[2]); (* increment destination *)
	BytesToClear:=BytesToClear -1; (* decrement number of bytes to copy *)
END_WHILE

END_FUNCTION

// Utils Functions/DELAYRETRY
FUNCTION_BLOCK DELAYRETRY
VAR_INPUT
	RETRIES	: BYTE:=5;
	DELAY	: TIME:=T#5S;
	(*TIMEOUT : TIME:=T#5s; (* Extend to support operation timeout *)*)
END_VAR
VAR_OUTPUT
	RUNNING : BOOL;
	EXEC	: BOOL; (* Execution semaphore *) 
	EV_ERR	: BOOL; (* Retries error *)
	EV_OK	: BOOL; (* Signal recovered state *)
END_VAR
VAR
	retry	: BYTE;
	tm1		: TON;	
END_VAR

EV_ERR:=FALSE;
EV_OK:=FALSE;

IF NOT (RUNNING OR EXEC) THEN
	IF retry=0 THEN EXEC:=TRUE;
	ELSE
		tm1(IN:=TRUE, PT:=DELAY); 
		IF tm1.Q THEN
			EXEC:=TRUE;
		END_IF
	END_IF
END_IF

ACTION Start:
RUNNING:=TRUE;
END_ACTION

ACTION Success:
RUNNING:=FALSE;
IF retry>=RETRIES THEN
	EV_OK:=TRUE;
END_IF
retry:=0;
EXEC:=TRUE;
END_ACTION

ACTION Fail:
RUNNING:=FALSE;
retry:=retry+1;
IF retry=RETRIES THEN
	EV_ERR:=TRUE;
END_IF
EXEC:=FALSE;
tm1(IN:=FALSE);
END_ACTION

END_FUNCTION_BLOCK

// Utils Functions/RAW16TOHEXSTR
FUNCTION RAW16TOHEXSTR : STRING(128)
VAR_INPUT
	pData: POINTER TO BYTE;
	DataLen: BYTE;
END_VAR
VAR
	pt: POINTER TO BYTE;
	xl: BYTE;
END_VAR

pt:=ADR(RAW16TOHEXSTR);
xl:=0;

WHILE DataLen>0 AND xl<120 DO

	pData:=pData+1;

	pt^ := (pData^ / 16#10) + 48 + (((pData^ / 16#10)/10)*7);
	pt:=pt+1;
	pt^ := (pData^ AND 16#0F)  + 48 + (((pData^ AND 16#0F)/10)*7);
	pt:=pt+1;

	pData:=pData-1;

	pt^ := (pData^ / 16#10) + 48 + (((pData^ / 16#10)/10)*7);
	pt:=pt+1;
	pt^ := (pData^ AND 16#0F)  + 48 + (((pData^ AND 16#0F)/10)*7);
	pt:=pt+1;

	xl:=xl+4;

	DataLen:=DataLen-2;
	pData:=pData+2;

END_WHILE

pt^:=0;

END_FUNCTION

// Utils Functions/RAWTOHEXSTR
FUNCTION RAWTOHEXSTR : STRING(128)
VAR_INPUT
	pData: POINTER TO BYTE;
	DataLen: BYTE;
END_VAR
VAR
	pt: POINTER TO BYTE;
	xl: BYTE;
END_VAR

pt:=ADR(RAWTOHEXSTR);

xl:=2;

WHILE DataLen>0 AND xl<128 DO

	pt^ := (pData^ / 16#10) + 48 + (((pData^ / 16#10)/10)*7);
	pt:=pt+1;
	pt^ := (pData^ AND 16#0F)  + 48 + (((pData^ AND 16#0F)/10)*7);
	pt:=pt+1;

	xl:=xl+2;

	DataLen:=DataLen-1;
	pData:=pData+1;

END_WHILE

pt^:=0;

END_FUNCTION

// Utils Functions/TONOF
FUNCTION_BLOCK TONOF
VAR_INPUT
	IN		: BOOL;
	PT_ON	: TIME; (* time to pass, before OUT is set *)
	PT_OF	: TIME; (* time to pass, before OUT is reset *)
END_VAR
VAR_OUTPUT
	OUT		: BOOL;
END_VAR
VAR
	timer	: TON;
END_VAR

IF IN<>OUT THEN
	timer(IN:=TRUE,PT:=SEL(IN,PT_OF,PT_ON));
	IF timer.Q THEN OUT:=IN; END_IF
ELSE
	timer(IN:=FALSE);
END_IF

END_FUNCTION_BLOCK

// Utils Functions/ADR_AT_INT
FUNCTION ADR_AT_INT : INT
VAR_INPUT
	ADDRESS : POINTER TO INT;
END_VAR
VAR
END_VAR

ADR_AT_INT:=ADDRESS^;

END_FUNCTION

// Plant_obj/obj_ASI
FUNCTION_BLOCK obj_ASI
(* === ASi INTERFACE ===
   v0.0[21/05/15] - Creation
*)
VAR_INPUT
	(* Settings *)
	ID				: BYTE;
	Refresh_Period	: TIME:=T#3M;
	Address			: BYTE;
	(* Controls *)
	Refresh_Auto	: BOOL:=TRUE; (* Enable automatic refresh *)
	Refresh_Now		: BOOL; 	  (* Force an immediate refresh *)
	(* Interface *)
	aPHY    : Get_ASi_PHY_Dat;
	aLCE    : Get_LCE;
	aLCEMS  : Get_LCEMS;
	aLPF	: Get_LPF;
	
END_VAR
VAR_OUTPUT
	(* Status *)
	Status_Log	: BYTE;
	Status_Vis	: DWORD;
END_VAR
VAR
	dly 	 	: TON := (PT:=T#5S);
	err 		: BYTE;
	err_old		: BYTE:=0;
	x			: byte;
	Tempor, Tempor1		: dword;
	Asi_Status_LCE, Asi_Status_LCEMS, Asi_Status_LPF : dword;
	Asi_DeviceA	: array[0..31] of bool;
	Asi_DeviceB	: array[0..31] of bool;
END_VAR
VAR_STAT
	Asi_DeviceAMem: array[0..31] of bool;
	Asi_DeviceBMem: array[0..31] of bool;	
END_VAR

(* Auto refresh timer *)
dly(IN:=NOT (dly.Q OR Refresh_Now OR (NOT Refresh_Auto)));
IF dly.Q THEN dly.PT:=Refresh_Period; Refresh_Now:=TRUE; END_IF

(* execute diagnostics *)
aPHY  (xExecute:=NOT Refresh_Now, enASi_Master:=SEL(ID=2,Master_1,Master_2));
aLCE  (xExecute:=NOT Refresh_Now, enASi_Master:=aPHY.enASi_Master);
aLCEMS(xExecute:=NOT Refresh_Now, enASi_Master:=aPHY.enASi_Master);
aLPF  (xExecute:=NOT Refresh_Now, enASi_Master:=aPHY.enASi_Master);
Refresh_Now:=FALSE;

(* Check status *)
IF aPHY.xReady AND aLCE.xReady AND aLCEMS.xReady AND aLPF.xReady THEN

	IF aPHY.xSE AND aPHY.xEF THEN err:=1;
	ELSIF aPHY.xPF1 THEN err:=2;
	ELSIF aPHY.xPF2 THEN err:=3;
	ELSIF aLCE.dwLCE_SA_Slaves<>0 OR aLCE.dwLCE_B_Slaves<>0 THEN err:=4;
	ELSIF aLCEMS.dwLCEMS_SA_Slaves<>0 OR aLCEMS.dwLCEMS_B_Slaves<>0 THEN err:=5;
	ELSIF aLPF.dwLPF_SA_Slaves<>0 OR aLPF.dwLPF_B_Slaves<>0 THEN err:=6;
	ELSE err:=0; END_IF
	
//Eseguo la scansione dei dati relativi alla rete asi e memorizzo lo stato di ogni indirizzo 
//negli array Asi_DeviceA e Asi_DeviceB. Questi dati verranno usati per la visualizzazione dello stato
//del nodo su PLC_visualization e verranno inoltrati al log.
	for x:=1 to 31 do
		Asi_Status_LCE := aLCE.dwLCE_B_Slaves and shl(1, x);
		Asi_Status_LCEMS := aLCEMS.dwLCEMS_B_Slaves and shl(1, x);
		Asi_Status_LPF := aLPF.dwLPF_SA_Slaves and shl(1, x);
		if (Asi_Status_LCE <> 0) or (Asi_Status_LCEMS <> 0)
			then Asi_DeviceB[x]:= TRUE;		
			else Asi_DeviceB[x]:= FALSE;
		end_if
	end_for

	for x:=0 to 31 do
		Asi_Status_LCE := aLCE.dwLCE_SA_Slaves and shl(1, x);
		Asi_Status_LCEMS := aLCEMS.dwLCEMS_SA_Slaves and shl(1, x);
		Asi_Status_LPF := aLPF.dwLPF_B_Slaves and shl(1, x);
		if (Asi_Status_LCE <> 0) or (Asi_Status_LCEMS <> 0)
			then Asi_DeviceA[x]:= TRUE;
			else Asi_DeviceA[x]:= FALSE;
		end_if
	end_for

	//gestione del log e inoltro del cambio di stato di un indirizzo asi, da fault a ready e viceversa
	//le informazioni vengono inoltrate al log e alla visualizzazione
	IF err<>err_old THEN
		err_old:=err;
		CASE err OF
			0: LogEv(EL_Log,EO_ASGW,ID,1,'ASi_OK');
					for x:=0 to 31 do
						 if (Asi_DeviceAMem [x] = TRUE) and (Asi_DeviceA[x] = FALSE) then
							 Asi_DeviceAMem [x] := FALSE;
							 case ID of
								 1: Address:=x;
								 2: Address:=x+63;
							 end_case
							 LogEv(EL_Log,EO_ASCBI,Address,3,'ASi_SLAVE_A_OK');
						 end_if	
					end_for
					for x:=1 to 31 do
						 if (Asi_DeviceBMem [x] = TRUE) and (Asi_DeviceB[x] = FALSE) then
							 Asi_DeviceBMem [x] := FALSE;
							 case ID of
								 1: Address:=x+32;
								 2: Address:=x+95;
							 end_case
							 LogEv(EL_Log,EO_ASCBI,Address,3,'ASi_SLAVE_B_OK');
						 end_if	
					end_for
			1,2,3: LogEv(EL_Alarm,EO_ASGW,ID,3,'ASi_ERR');
					for x:=0 to 31 do
						 if (Asi_DeviceAMem [x] = TRUE) and (Asi_DeviceA[x] = FALSE) then
							 Asi_DeviceAMem [x] := FALSE;
							 case ID of
								 1: Address:=x;
								 2: Address:=x+63;
							 end_case
							 LogEv(EL_Log,EO_ASCBI,Address,3,'ASi_SLAVE_A_OK');
						 end_if	
					end_for
					for x:=1 to 31 do
						 if (Asi_DeviceBMem [x] = TRUE) and (Asi_DeviceB[x] = FALSE) then
							 Asi_DeviceBMem [x] := FALSE;
							 case ID of
								 1: Address:=x+32;
								 2: Address:=x+95;
							 end_case
							 LogEv(EL_Log,EO_ASCBI,Address,3,'ASi_SLAVE_B_OK');
						 end_if	
					end_for
			4,5,6:
					LogEv(EL_Wrn,EO_ASGW,ID,2,'ASi_SLAVE_ERR');
					for x:=0 to 31 do
						 if Asi_DeviceA[x] = TRUE then
							 Asi_DeviceAMem [x] := TRUE;
							 case ID of
								 1: Address:=x;
								 2: Address:=x+63;
							 end_case
							 LogEv(EL_Alarm,EO_ASCBI,Address,3,'ASi_SLAVE_A_ERR');
						 end_if	
					end_for
					for x:=1 to 31 do
						 if Asi_DeviceB[x] = TRUE then	
							 Asi_DeviceBMem [x] := TRUE;
							 case ID of
								 1: Address:=x+32;
								 2: Address:=x+95;
							 end_case
							LogEv(EL_Alarm,EO_ASCBI,Address,3,'ASi_SLAVE_B_ERR');
						end_if
					end_for
		END_CASE
	END_IF

	(* Log/visu status *)
	   IF err>0  AND err<4 THEN Status_Log:=2; Status_Vis:=COLOR_RED;
	ELSIF err>=4           THEN Status_Log:=1; Status_Vis:=COLOR_YELLOW;
					 	   ELSE Status_Log:=0; Status_Vis:=COLOR_GREEN;
	END_IF

END_IF

END_FUNCTION_BLOCK

// Plant_obj/obj_CRON
FUNCTION_BLOCK obj_CRON
(* === CRONOGRAFO STANDARD ===
   v1.0[16/04/05] - Versioning
*)
VAR_INPUT
	(* Settings *)
	ID			: WORD;	//BYTE;		(* Index of instanced object *)

	InitOK		: BOOL;
	Alarm		: BOOL;
	Warning		: BOOL;

	Profile		: typ_Cron_Profile; 				(* Profilo attivo *)
	ProfileNr	: BYTE;								(* Indice profilo attivo *)
	CalendarIdx : WORD;								(* Indice calendario attivo *)
	Jolly		: ARRAY[0..9] OF typ_Cron_Jolly;	(* Jolly attivi *)
	
	SET_POINT		: INT;	//GIURE ver 21
	(* Status *)
	STAT_LOG		: BYTE; //GIURE ver 21

END_VAR
VAR_IN_OUT
END_VAR
VAR_OUTPUT
	SetPoint		: INT;
	(* Status *)
	Status_Log		: BYTE;
	Status_Vis 		: DWORD;
END_VAR
VAR
	Buf: 	ARRAY[0..512] OF BYTE;
	hFile		: RTS_IEC_HANDLE;
	hRes		: RTS_IEC_RESULT;
	sFile: 	STRING;
	sFile2: STRING;

	i:		WORD;
	t1:		DWORD;
	t2:		BOOL;

END_VAR

(* Check initialization *)
IF NOT 
	InitOK 
THEN 
	Init(); 
END_IF

(* Chrono *)
IF CalendarIdx<>Sys.Time_CT_Day THEN DB_Load(); END_IF
SetPoint:=Profile.Setpoint[Sys.Time_CT_Quarter];

(* Check jolly *)
FOR i := 0 TO 9 DO
	IF ( DT_TO_DWORD(Jolly[i].Start)>0  AND Jolly[i].End>Jolly[i].Start AND
	     Jolly[i].Start<=Sys.Time_CT_DT AND Jolly[i].End>Sys.Time_CT_DT ) THEN
			SetPoint:=Jolly[i].Temp;
	END_IF
END_FOR


(* Status color *)
   IF Alarm   THEN Status_Log:=2; Status_Vis:=16#2020F0;
ELSIF Warning THEN Status_Log:=1; Status_Vis:=16#20F0F0;
              ELSE Status_Log:=0; Status_Vis:=COLOR_GREEN;	//16#20F020;
			  END_IF

ACTION DB_Create:
(*(* Check presence of previous year *)
sFile2:=REPLACE(STR1:=sFile, STR2:=WORD_TO_STRING(Sys.Time_Year-1), L:=4, P:=LEN(FilesPath)+1);
hFile:=SysFileOpen(sFile2, AM_READ, ADR(hRes));
IF hFile<>RTS_INVALID_HANDLE THEN
	(* Check file version and close *)
	SysFileRead(hFile, ADR(Buf), 1, ADR(hRes));
	SysFileClose(hFile);
END_IF
IF hFile<>RTS_INVALID_HANDLE AND Buf[0]=1 THEN
	(* Copy file *)
	SysFileCopy(sFile, sFile2);
ELSE*)
	(* Create empty file *)
	hFile:=SysFileOpen(sFile, AM_WRITE, ADR(hRes));
	MEMCLR(pDestinationAddress:=ADR(Buf), BytesToClear:=SIZEOF(Buf));
	FOR i := 0 TO 10239 BY 512 DO
		SysFileWrite(hFile, ADR(Buf), 512, ADR(hRes));
	END_FOR
	Buf[0]:=1;
	SysFileSetPos(hFile, 0);
	SysFileWrite(hFile, ADR(Buf), 1, ADR(hRes));
	SysFileClose(hFile);
//END_IF
END_ACTION

ACTION DB_Load:
DB_SetName();

(* Open data file *)
hFile:=SysFileOpen(sFile, AM_READ, ADR(hRes));

(* File not found *)
IF hFile=RTS_INVALID_HANDLE THEN
	Warning:=TRUE;
	LogEv(EL_Wrn,EO_CRON,ID,1,'No_data_file');
	DB_Create();
	(* Reopen file *)
	hFile:=SysFileOpen(sFile, AM_READ, ADR(hRes));
	IF hFile=RTS_INVALID_HANDLE THEN
		Alarm:=TRUE;
		LogEv(EL_Alarm,EO_CRON,ID,3,'Filesystem_error');
		RETURN;
	END_IF
END_IF

(* Check version *)
SysFileRead(hFile, ADR(Buf), 1, ADR(hRes));
IF Buf[0]<>1 THEN
	IF NOT Alarm THEN
		Alarm:=TRUE;
		LogEv(EL_Alarm,EO_CRON,ID,2,'Bad_data_version');
	END_IF
	SysFileClose(hFile);
	RETURN;
END_IF

(* Read Jolly data *)
SysFileSetPos(hFile, 512);
SysFileRead(hFile, ADR(Jolly), SIZEOF(Jolly), ADR(hRes));
(* Read active profile index *)
CalendarIdx:=Sys.Time_CT_Day;
SysFileSetPos(hFile, (1024+4*CalendarIdx));
SysFileRead(hFile, ADR(ProfileNr), SIZEOF(ProfileNr), ADR(hRes));
(* Read active profile *)
SysFileSetPos(hFile, (3072+512*ProfileNr));
SysFileRead(hFile, ADR(Profile), SIZEOF(Profile), ADR(hRes));

(* Close file and validate data *)
SysFileClose(hFile);
END_ACTION

ACTION DB_SetName:
(* Create current filename 'yyyyCRnn.DAT' *)
sFile:=CONCAT(ConfPath,WORD_TO_STRING(Sys.Time_Year));
sFile:=CONCAT(STR1:=sFile, STR2:='CR');
IF ID<10 THEN
sFile:=CONCAT(STR1:=sFile, STR2:='0');
END_IF
//sFile:=CONCAT(STR1:=sFile, STR2:=BYTE_TO_STRING(ID));
sFile:=CONCAT(STR1:=sFile, STR2:=WORD_TO_STRING(ID));
sFile:=CONCAT(STR1:=sFile, STR2:='.DAT');
END_ACTION

ACTION Init:
DB_Load();
InitOK:=TRUE;
END_ACTION

ACTION AddLogData:
//Genera la stringa di log dei cronografi	//GIURE ver 21
//Logger.s1:=INSERT('&CRON=',BYTE_TO_STRING(ID),5);
Logger.s1:=INSERT('&CRON=',WORD_TO_STRING(ID),5);
IF ID<10 THEN Logger.s1:=INSERT(Logger.s1,'0',5); END_IF

Logger.s1:=CONCAT(Logger.s1,INT_TO_STRING(SET_POINT));		
Logger.s1:=CONCAT(Logger.s1,';');
Logger.s1:=CONCAT(Logger.s1,BYTE_TO_STRING(STAT_LOG));
ADDSTRING(ADR(Logger.TData), ADR(Logger.s1), Logger.TLen);
END_ACTION

END_FUNCTION_BLOCK

// Plant_obj/obj_CRON_EDITOR
FUNCTION_BLOCK obj_CRON_EDITOR
(* === EDITOR CRONOGRAFO ===
   v1.0[16/04/05] - Versioning
*)
VAR_INPUT

	(* Common selections *)
	CN_Sel:			BYTE:=1;
	CN_Act:			word;	//BYTE;
	CN_YSel:		WORD:=2016;
	CN_YAct:		WORD;

	(* Profile editor *)
	PR_Sel: 		BYTE:=1;
	PR_Act:			BYTE;
	PR_TT:			REAL;
	PR:				typ_Cron_Profile;
	(* Profile signals *)
	PR_Load:		BOOL;
	PR_Save:		BOOL;

	(* Calendar editor *)
	CA_Sel:			BYTE:=1; (* Calendar month selected *)
	CA_Act:			BYTE;    (* Calendar month active *)
	CA_DayF:		BYTE:=0;
	CA_DayL:		BYTE:=31;
	CA_TPR:			BYTE;
	CA:				typ_Cron_Calendar; (* Only used for first 32 entries *)
	(* Calendar signals *)
	CA_Load:		BOOL;
	CA_Save:		BOOL;

	(* Jolly editor *)
	JL:				ARRAY[0..9] OF typ_Cron_Jolly;
	(* Jolly signals *)
	JL_Load:		BOOL;
	JL_Save:		BOOL;

	Invisible:		bool;
END_VAR
VAR_OUTPUT
	Message		: STRING;
END_VAR
VAR
	sFileName	: STRING;
	hMode		: ACCESS_MODE;
	hFile		: RTS_IEC_HANDLE;
	hRes		: RTS_IEC_RESULT;
	x			: word;
	i			: WORD;
	ver			: BYTE;
	r1			: BOOL;
	r2			: DWORD;

END_VAR

for x:= 1 to CRON_MAX do
	if CRON[x].ID = CronEd.CN_Sel then
		CN_Act:=x;
		Invisible := FALSE;
		exit;	
		else
			Invisible := TRUE;
	end_if
end_for


IF PR_Load 
	THEN 
		PR_Load_Exe(); 
		PR_Load:=FALSE; 
END_IF
IF PR_Save 
	THEN 
		PR_Save_Exe(); PR_Save:=FALSE; 
END_IF
IF CA_Load 
THEN 
	CA_Load_Exe(); CA_Load:=FALSE; 
END_IF
IF CA_Save 
THEN 
	CA_Save_Exe(); CA_Save:=FALSE; 
END_IF
IF JL_Load 
	THEN 
	JL_Load_Exe(); JL_Load:=FALSE; 
END_IF
IF JL_Save 
	THEN 
	JL_Save_Exe(); JL_Save:=FALSE; 
END_IF

ACTION CA_Load_Exe:
hMode:=AM_READ;
FileOpen();

IF hFile<>RTS_INVALID_HANDLE THEN

	(* Read calendar month *)
	FOR i := 0 TO 31 DO
		SysFileSetPos(hFile, (1024 + ((CA_Sel-1)*32 + i)*4) );
		SysFileRead(hFile, ADR(CA.Profile[i]), 1, ADR(hRes));
	END_FOR

	(* Close file *)
	SysFileClose(hFile);

	(* Validate data *)
	CA_Act :=CA_Sel;
	//CN_Act :=CN_Sel;
	CN_YAct:=CN_YSel;

	Message:='Calendar load OK';

END_IF
END_ACTION

ACTION CA_Save_Exe:
hMode:=AM_READ_PLUS;
FileOpen();

IF hFile<>RTS_INVALID_HANDLE THEN

	(* Write calendar month *)
	FOR i := 0 TO 31 DO
		SysFileSetPos(hFile, (1024 + ((CA_Sel-1)*32 + i)*4) );
		SysFileWrite(hFile, ADR(CA.Profile[i]), 1, ADR(hRes));
	END_FOR

	(* Close file *)
	SysFileClose(hFile);

	Message:='Calendar save OK';

END_IF
END_ACTION

ACTION FileOpen:
(* Create current filename 'yyyyCRnn.DAT' *)
sFileName:=CONCAT(ConfPath,WORD_TO_STRING(CN_YSel));
sFileName:=CONCAT(STR1:=sFileName, STR2:='CR');
IF CN_Sel<10 THEN
sFileName:=CONCAT(STR1:=sFileName, STR2:='0');
END_IF
sFileName:=CONCAT(STR1:=sFileName, STR2:=BYTE_TO_STRING(CN_Sel));
sFileName:=CONCAT(STR1:=sFileName, STR2:='.DAT');

(* Check file version and size! *)
(* ... *)

(* Open data file *)
hFile:=SysFileOpen(sFileName,AM_READ,ADR(hRes));

(* File not found *)
IF hFile=RTS_INVALID_HANDLE THEN
	Message:='File not found';
	RETURN;
END_IF

(* Close file *)
SysFileClose(hFile);

(* Open data file *)
hFile:=SysFileOpen(sFileName,hMode,ADR(hRes));
END_ACTION

ACTION JL_Load_Exe:
hMode:=AM_READ;
FileOpen();

IF hFile<>RTS_INVALID_HANDLE THEN

	(* Read jolly *)
	SysFileSetPos(hFile, 512);
	SysFileRead(hFile, ADR(JL), SIZEOF(JL), ADR(hRes));

	(* Close file *)
	SysFileClose(hFile);

	(* Validate data *)
	//CN_Act:=CN_Sel; //GIURE modifica per AF Principale
	CN_YAct:=CN_YSel;

	Message:='Jolly load OK';

END_IF
END_ACTION

ACTION JL_Save_Exe:
hMode:=AM_READ_PLUS;
FileOpen();

IF hFile<>RTS_INVALID_HANDLE THEN

	(* Write selected profile *)
	SysFileSetPos(hFile, 512);
	SysFileWrite(hFile, ADR(JL), SIZEOF(JL), ADR(hRes));

	(* Close file *)
	SysFileClose(hFile);

	Message:='Jolly save OK';

END_IF
END_ACTION

ACTION PR_Load_Exe:
hMode:=AM_READ;
FileOpen();

IF hFile<>RTS_INVALID_HANDLE THEN

	(* Read selected profile *)
	SysFileSetPos(hFile, (3072 + 512*PR_Sel));
	SysFileRead(hFile, ADR(PR), SIZEOF(PR), ADR(hRes));

	(* Close file *)
	SysFileClose(hFile);
	(*
	for x:= 1 to CRON_MAX do
		if LuxElement[x].ID = CronEd.CN_Sel then
			CN_Act:=x;	
			x:= CRON_MAX;
		end_if
	end_for
	*)
	(* Validate data *)
	PR_Act:=PR_Sel;
	//CN_Act:=CN_Sel; //GIURE modifica per AF Principale
	CN_YAct:=CN_YSel;

	Message:='Profile load OK';

END_IF
END_ACTION

ACTION PR_Save_Exe:
hMode:=AM_READ_PLUS;
FileOpen();

IF hFile<>RTS_INVALID_HANDLE THEN

	(* Write selected profile *)
	SysFileSetPos(hFile, (3072 + 512*PR_Sel));
	SysFileWrite(hFile, ADR(PR), SIZEOF(PR), ADR(hRes));

	(* Close file *)
	SysFileClose(hFile);

	Message:='Profile save OK';

END_IF
END_ACTION

END_FUNCTION_BLOCK

// Plant_obj/obj_PSG_old
FUNCTION_BLOCK obj_PSG_old
(* === Passage sensor ===
   v1.0[27/05/15] - Create
*)
VAR_INPUT
	(* Settings *)
	ID				: BYTE;
	xPolarity		: BOOL:=TRUE;  (* Default unoccupied polarity *)
	TimErr_timeout	: TIME:=T#30M; (* Timeout for occupied barrier error *)
(*	WRN_TIMEOUT		: TIME:=T#5M;  (* Timeout fot occupied barrier warning *)*)	
(*	ACT_TIMEOUT 	: TIME:=T#7D;  (* Timeout for inactive barrier warning *)*)
(*	DISTANCE		: WORD; 	   (* Distance to 2th sensor in mm *)*)
(*  SPEED_THRESHOLD : INT;         (* Speed threshold for output trigger *)*)
	(* Ack output events *)
	xSense_trig		: BOOL;
(*	SPEED_TRIG		: BOOL; *)
	(* Physical inputs *)
	PSG_IN			: BOOL;        (* Sensor input *)
(*	PSG_IN2			: BOOL;        (* Optional speed input sensor *)*)	
END_VAR
VAR_IN_OUT
	PASSAGES		: DWORD;
(*	SPEED			: AVERAGE_INT; *)	
END_VAR
VAR_OUTPUT
	xSensor			: BOOL;	//set a 1 sul fronte di salita della fotocellula corrispondente
	(* Status *)
	Status_Log		: BYTE;
	Status_Vis 		: DWORD;
END_VAR
VAR
	evnt	: FLT_EVENT;
	errt	: TON;
	errtev	: FLT_EVENT;

(*	wrnt	: TON;*)
(*	actt	: TON:*)
END_VAR

xSensor:=PSG_IN XOR xPolarity;	//Default: PSG_IN normalmente true, xPolarity = True --> xSensor = False
								//In presenza di attivazione del passaggio: PSG_IN = false, xPolarity = True --> xSensor = True
(* Statistics *)
evnt(IN:=xSensor);
IF evnt.EVH THEN
	xSense_trig:=TRUE;
	IF PASSAGES=16#FFFFFFFF THEN
		LogEv(EL_Wrn,EO_PSG,ID,5,'');
		PASSAGES:=1;
	ELSE
		PASSAGES:=PASSAGES+1;
	END_IF
END_IF

(* Error check *)
errt(IN:=xSensor, PT:=TimErr_timeout);
errtev(IN:=errt.Q);
IF errtev.EVH THEN
	Status_Log:=2; Status_Vis:=COLOR_RED;
	LogEv(EL_Alarm,EO_PSG,ID,2,'');
END_IF
IF errtev.EVL THEN
	Status_Log:=0; Status_Vis:=COLOR_GREEN;
	LogEv(EL_Log,EO_PSG,ID,1,'');
END_IF

ACTION StatReset:
(* Reset statistic counters *)
PASSAGES:=0;
END_ACTION

END_FUNCTION_BLOCK

// Plant_obj/obj_LUXM_old
FUNCTION_BLOCK obj_LUXM_old
(* === Metered ON/OFF Illumination Point ===
   Failure detection:
   Statistic data:
   
   - Come identifico l'assenza del nodo?? (Rele non funzionante/non alimentato)
   - Acquisizione carico dopo accensione?? Dati carico in NVM!
   
   v1.0[07/05/15] - Create
*)
VAR_INPUT
	(* Settings *)
	ID				: BYTE;
	(* Controls *)
	CTRL_MODE		: INT:=100;  (* 0:MAN OFF, -1:MAN-ON,
							   -2:KEY-ON, -3:KEY-OFF, -4:DAY, -5:NIGHT,
							   N>0:Nsec-TIMER *)
	CTRL_TRIG		: BOOL; (* Trigger for timer start *)
	CTRL_KEY		: BOOL; (* External KEY control input *)
	CTRL_SENS		: BOOL; (* External dark sensor input [1:Dark] *)
	CTRL_EXTON		: BOOL; (* External forced activation *)
	(* Physical inputs *)
	REL_ST			: BOOL; (* Status feedback *)
	REL_V			: WORD; (* [E-1 V] Voltage *)
	REL_A			: WORD; (* [E-1 A] Current *)
	REL_ALM			: WORD; (* Error status [0:OK, 1:Disconnected, 2:LoadLOW, 3:LoadHIGH, 4:Overload, 5:ControlFAIL] *)
	REL_TEMP		: INT;  (* [E-1 °C] Temperature *)
	REL_TON			: DWORD;(* [sec] External working time counter *)  
	(* Persistent *)(*
	WORKINGTIME		: POINTER TO DWORD; (* [sec] Internal working time counter *)
	POWERONCYCLES	: POINTER TO DWORD; (* Internal counter of power-on cycles *)
	ENERGYCOUNTER	: POINTER TO DWORD; (* [E-1 kWh] Internal energy counter *)
	ENERGYCOUNTER_T : POINTER TO DWORD; (* Temporary energy in E-2*Wsec *)*)
	PressKeyVisuOn	: BOOL := 0;
	PressKeyVisuOff	: BOOL := 0;
END_VAR
VAR_IN_OUT
//VAR_OUTPUT RETAIN PERSISTENT
	WORKINGTIME		: DWORD; (* [sec] Internal working time counter *)
	POWERONCYCLES	: DWORD; (* Internal counter of power-on cycles *)
	ENERGYCOUNTER	: DWORD; (* [E-1 kWh] Internal energy counter *)
	ENERGYCOUNTER_T : DWORD; (* Temporary energy in E-2*Wsec *)
END_VAR
VAR_OUTPUT
	(* Physical outputs *)
	REL_EN			: BOOL;	(* Control output *)
	(* Status *)
	Status_Log		: BYTE;
	Status_Vis 		: DWORD;
END_VAR
VAR
	TickTimer		: TON := ( PT:=T#1S );
	TrigTimer		: TOF;
	sREL_EN			: FLT_EVENT;
	sREL_ALM		: WORD:=16#FFFF;
	chkREL_ST		: FLT_TIME := ( TTAP:=T#20S, INITEV:=FALSE );
END_VAR

(* Trig timer *)
TrigTimer(IN:=CTRL_TRIG);

(* Control logic *)
IF CTRL_EXTON THEN
	REL_EN:=TRUE;
ELSE
	CASE CTRL_MODE OF
		 0: REL_EN:=FALSE;
		-1: REL_EN:=TRUE;
		-2: REL_EN:=CTRL_KEY;
		-3: REL_EN:=NOT CTRL_KEY;
		-4: REL_EN:=CTRL_SENS;
		-5: REL_EN:=NOT CTRL_SENS;
	ELSE
		IF CTRL_MODE>0 THEN
			REL_EN:=TrigTimer.Q;
			TrigTimer.PT:=T#1S*CTRL_MODE;
		ELSE
			REL_EN:=FALSE;
		END_IF
	END_CASE
END_IF

(* Temporary energy counter *)
TickTimer(IN:=NOT TickTimer.Q);
IF TickTimer.Q AND REL_EN THEN
	WORKINGTIME:=WORKINGTIME+1;
	ENERGYCOUNTER_T:=ENERGYCOUNTER_T+REL_V*REL_A;
	IF ENERGYCOUNTER_T>36000000 THEN
		ENERGYCOUNTER_T:=ENERGYCOUNTER_T-36000000;
		ENERGYCOUNTER:=ENERGYCOUNTER+1;		
	END_IF
END_IF

(* Generate status events *)
sREL_EN(IN:=REL_EN);
IF sREL_EN.EVL THEN LogEv(EL_Log,EO_LUXM,ID,2,''); END_IF
IF sREL_EN.EVH THEN LogEv(EL_Log,EO_LUXM,ID,3,''); POWERONCYCLES:=POWERONCYCLES+1; END_IF

(* Check status feedback *)
chkREL_ST(IN:=(REL_ST<>REL_EN));
IF chkREL_ST.EVH THEN LogEv(EL_Alarm,EO_LUXM,ID,9,''); END_IF
IF chkREL_ST.EVL AND sREL_ALM=0 THEN LogEv(EL_Log,EO_LUXM,ID,1,''); END_IF

(* Check controller alarm *)
IF sREL_ALM<>REL_ALM THEN
	CASE REL_ALM OF
		0: IF NOT chkREL_ST.OUT THEN LogEv(EL_Log,EO_LUXM,ID,1,''); END_IF
		1: LogEv(EL_Alarm,EO_LUXM,ID,6,'');
		2: LogEv(EL_Wrn  ,EO_LUXM,ID,4,WORD_TO_STRING(REL_A));
		3: LogEv(EL_Wrn  ,EO_LUXM,ID,5,WORD_TO_STRING(REL_A));
		4: LogEv(EL_Alarm,EO_LUXM,ID,7,WORD_TO_STRING(REL_A));
		5: LogEv(EL_Alarm,EO_LUXM,ID,8,'');
	END_CASE
	sREL_ALM:=REL_ALM;
END_IF

(* Status color *)
   IF REL_ALM=1 OR REL_ALM>3 OR chkREL_ST.OUT	THEN Status_Log:=2; Status_Vis:=COLOR_RED;
ELSIF REL_ALM<>0								THEN Status_Log:=1; Status_Vis:=COLOR_YELLOW;
                  	   							ELSE Status_Log:=0; Status_Vis:=SEL(REL_EN,COLOR_GREEN_OFF,COLOR_GREEN);
END_IF

ACTION AddLogData:
Logger.s1:=INSERT('&LUXM=',BYTE_TO_STRING(ID),5);
IF ID<10 THEN Logger.s1:=INSERT(Logger.s1,'0',5); END_IF

Logger.s1:=CONCAT(Logger.s1,WORD_TO_STRING(REL_V));				Logger.s1:=CONCAT(Logger.s1,';');
Logger.s1:=CONCAT(Logger.s1,WORD_TO_STRING(REL_A));				Logger.s1:=CONCAT(Logger.s1,';');
Logger.s1:=CONCAT(Logger.s1,DWORD_TO_STRING(ENERGYCOUNTER));	Logger.s1:=CONCAT(Logger.s1,';');
Logger.s1:=CONCAT(Logger.s1,DWORD_TO_STRING(WORKINGTIME));		Logger.s1:=CONCAT(Logger.s1,';');
Logger.s1:=CONCAT(Logger.s1,DWORD_TO_STRING(POWERONCYCLES));	Logger.s1:=CONCAT(Logger.s1,';');
Logger.s1:=CONCAT(Logger.s1,INT_TO_STRING(REL_TEMP));			Logger.s1:=CONCAT(Logger.s1,';');

Logger.s1:=CONCAT(Logger.s1,BYTE_TO_STRING(Status_Log));
ADDSTRING(ADR(Logger.TData), ADR(Logger.s1), Logger.TLen);
END_ACTION

ACTION StatReset:
(* Reset statistic counters *)
WORKINGTIME:=0;
POWERONCYCLES:=0;
ENERGYCOUNTER:=0;
END_ACTION

END_FUNCTION_BLOCK

// Utils Functions/GenerateTabs
FUNCTION GenerateTabs : BOOL
VAR_INPUT
END_VAR
VAR
END_VAR

(*
	TabASI1AB_FromFile	: ARRAY [1..31] OF BYTE;
	TabASI1Add_FromFile	: ARRAY [1..31] OF BYTE;
	TabASI1BitAdd_FromFile	: ARRAY [1..31] OF BYTE;
	TabASI1PSG_FromFile	: ARRAY [1..31] OF WORD;
	
	ASI_1	 : ARRAY [ASI_A..ASI_B,1..31,0..3] OF BOOL;
	ASI_2	 : ARRAY [ASI_A..ASI_B,1..31,0..3] OF BOOL;
	PSG_LIST : ARRAY [1..PSG_MAX] OF BOOL;
*)

TabASI1AB_FromFile[1] := ASI_A;
TabASI1Add_FromFile[1] := 1;
TabASI1BitAdd_FromFile[1] := 0;
TabASI1PSG_FromFile[1] := 89;

TabASI1AB_FromFile[2] := ASI_A;
TabASI1Add_FromFile[2] := 1;
TabASI1BitAdd_FromFile[2] := 2;
TabASI1PSG_FromFile[2] := 90;

ASI_1[TabASI1AB_FromFile[1], TabASI1Add_FromFile[1], TabASI1BitAdd_FromFile[1]] := PSG_LIST[TabASI1PSG_FromFile[1]];

ASI_1[TabASI1AB_FromFile[2], TabASI1Add_FromFile[2], TabASI1BitAdd_FromFile[2]] := PSG_LIST[TabASI1PSG_FromFile[2]];

END_FUNCTION

// Utils Functions/OpenFiles_ASI_PSG_FB_backup
//Esegue la lettura del file x_ASI_PSG.txt per poi configurare le tabelle ASI_1 e ASI_2 di associazione tra passaggi e segnali di input 
FUNCTION_BLOCK OpenFiles_ASI_PSG_FB_backup
VAR_INPUT
	//sFileName : STRING;
END_VAR
VAR_OUTPUT
	Message		: STRING;
END_VAR
VAR
	hMode		: ACCESS_MODE;
	hFile		: RTS_IEC_HANDLE;
	hRes		: RTS_IEC_RESULT;
	bList		: ARRAY [0..15] OF BYTE;
	i			: DWORD; //Dim max file: 2^32 byte
	j			: BYTE; //Indice dell'array bList
	k			: BYTE; //Indice tabella ASI 2^8 = 256
	xwDimFile	: LWORD;
	bChar		: BYTE;
	sFileName 	: STRING;
END_VAR

(* Create current filename 'yyyyCRnn.DAT' *)
//sFileName:=CONCAT(ConfPath,WORD_TO_STRING('2ASI_LUX.txt'));
//sFileName:=CONCAT(STR1:=sFileName, STR2:='CR');
//IF CN_Sel<10 THEN
//sFileName:=CONCAT(STR1:=sFileName, STR2:='0');
//END_IF
//sFileName:=CONCAT(STR1:=sFileName, STR2:=BYTE_TO_STRING(CN_Sel));
//sFileName:=CONCAT(STR1:=sFileName, STR2:='.DAT');
//sFileName:='/media/sd/2015CR01.DAT';	//2_ASI_LUX.txt';
(* Check file version and size! *)
(* ... *)

(* Open data file *)
sFileName:=CONCAT(STR1:=MapConf_Path, STR2:=PLC_ID);
sFileName:=CONCAT(STR1:=sFileName, STR2:=AsiPsg_FileName);
hFile:=SysFileOpen(sFileName,AM_READ,ADR(hRes));

(* File not found *)
IF hFile=RTS_INVALID_HANDLE THEN
	Message:='File not found';
	RETURN;
END_IF

(* Close file *)
SysFileClose(hFile);

(* Open data file *)
i:=0; //indice di scorrimento del file
j:=0; //indice di scorrimento dell'array dove viene momentaneamente memorizzata la riga prima del ;
k:=0; //indice della tabella di mappatura ASI
hFile:=SysFileOpen(sFileName,hMode,ADR(hRes));
WHILE SysFileEOF(hFile)<> 0 DO
	SysFileSetPos(hFile, i);	
	SysFileRead(hFile, ADR(bList[j]), 1, ADR(hRes));
	IF bList[j] = 16#2F  // se trovo '/'
		THEN 
			SysFileSetPos(hFile, i+1);	
			SysFileRead(hFile, ADR(bList[j+1]), 1, ADR(hRes));
			IF bList[j+1] = 16#2F  // se trovo ancora '/'
				THEN 
					WHILE  bList[j]<> 16#0D DO
						i := i+1;
						SysFileSetPos(hFile, i);	
						SysFileRead(hFile, ADR(bList[j]), 1, ADR(hRes));
					END_WHILE	
					i := i+1;
					SysFileSetPos(hFile, i);	
					SysFileRead(hFile, ADR(bList[j]), 1, ADR(hRes));
					IF bList[j] = 16#0A
						THEN 
							i := i+1;
							j := 0;
							SysFileSetPos(hFile, i);	
							SysFileRead(hFile, ADR(bList[j]), 1, ADR(hRes)); //leggo il primo carattere della nuova riga
						ELSE 
							Message:='Errore 0D 0A';
							RETURN;
					END_IF
				ELSE 
					Message:='Errore //';
					RETURN;
			END_IF
	END_IF
	IF bList[j] <> 16#3B //finchè non trovo ;
		THEN 
			i:=i+1;
			j:=j+1;	
		ELSE
			i:=i+3; //Se trovo ; inizio a salvare i dati della riga letta in TabAsiPsg[k]....
			j:=0;
			k:=k+1;
			TabAsiPsg[k].Asi1_2 := (bList[0]-16#30); //memorizzo se asi 1 o asi 2
			IF 	bList[4] = 16#41	//Se contiene il carattere A
				THEN TabAsiPsg[k].A_B := ASI_A;
				ELSE TabAsiPsg[k].A_B := ASI_B;
			END_IF		
			TabAsiPsg[k].Address :=  (bList[2]-16#30)*10 + (bList[3]-16#30); //memorizzo indirizzo
			TabAsiPsg[k].Bit_address := bList[6]-16#30;		//memorizzo il bit
			TabAsiPsg[k].PSG := (bList[8]-16#30)*100 + (bList[9]-16#30)*10 + (bList[10]-16#30); //memorizzo il passaggio associato
				
			(*		
			CASE bList[0] OF
			16#31:
				IF 	bList[4] = 16#41	//Se contiene il carattere A
					THEN TabASI1[k].A_B := ASI_A;
					ELSE TabASI1[k].A_B := ASI_B;
				END_IF		
				TabASI1[k].Address :=  (bList[2]-16#30)*10 + (bList[3]-16#30);
				TabASI1[k].Bit_address := bList[6]-16#30;
				TabASI1[k].PSG := (bList[8]-16#30)*100 + (bList[9]-16#30)*10 + (bList[10]-16#30);
				
			16#32:
				IF 	bList[4] = 16#41	//Se contiene il carattere A
					THEN TabASI2[k].A_B := ASI_A;
					ELSE TabASI2[k].A_B := ASI_B;
				END_IF		
				TabASI2[k].Address :=  (bList[2]-16#30)*10 + (bList[3]-16#30);
				TabASI2[k].Bit_address := bList[6]-16#30;
				TabASI2[k].PSG := (bList[8]-16#30)*100 + (bList[9]-16#30)*10 + (bList[10]-16#30);
		END_CASE 
			CASE bList[0] OF
			16#31:
				IF 	bList[4] = 16#41	//Se contiene il carattere A
					THEN TabASI1AB_FromFile[1] := ASI_A;
					ELSE TabASI1AB_FromFile[1] := ASI_B;
				END_IF		
				TabASI1Add_FromFile[1] :=  (bList[2]-16#30)*10 + (bList[3]-16#30);
				TabASI1BitAdd_FromFile[1] := bList[6]-16#30;
				TabASI1PSG_FromFile[1] := (bList[8]-16#30)*100 + (bList[9]-16#30)*10 + (bList[10]-16#30);
			16#32:
				IF 	bList[4] = 16#41	//Se contiene il carattere A
					THEN TabASI2AB_FromFile[1] := ASI_A;
					ELSE TabASI2AB_FromFile[1] := ASI_B;
				END_IF		
				TabASI2Add_FromFile[1] :=  (bList[2]-16#30)*10 + (bList[3]-16#30);
				TabASI2BitAdd_FromFile[1] := bList[6]-16#30;
				TabASI2PSG_FromFile[1] := (bList[8]-16#30)*100 + (bList[9]-16#30)*10 + (bList[10]-16#30);
		END_CASE *)
	END_IF	
END_WHILE
xwDimFile:=SysFileGetSize(sFileName,ADR(hRes));

END_FUNCTION_BLOCK

// Utils Functions/LuxEnable_FB
FUNCTION_BLOCK LuxEnable_FB
VAR_INPUT
END_VAR
VAR_OUTPUT
END_VAR
VAR
	wCounter: WORD;
END_VAR

FOR wCounter := 1 TO MAX_LUXNUM DO
	CASE TabDefaultLux[wCounter].Mode of
		0:	; //Spegnere perchè in manuale off
		1:	; //Accendere perchè in manuale on
		2:	; //Controllo timer da fotocellule
		3:	; //Cronografo
	END_CASE
END_FOR

END_FUNCTION_BLOCK

// Plant_obj/obj_LUXM_backUp
FUNCTION_BLOCK obj_LUXM_backUp
(* === Metered ON/OFF Illumination Point ===
   Failure detection:
   Statistic data:
   
   - Come identifico l'assenza del nodo?? (Rele non funzionante/non alimentato)
   - Acquisizione carico dopo accensione?? Dati carico in NVM!
   
   v1.0[07/05/15] - Create
*)
VAR_INPUT
	(* Settings *)
	ID				: BYTE;
	ptNextLux, ptPrevLux : POINTER TO obj_LUXM := 16#FFFFFFFF;
	(* Controls *)
	CTRL_MODE		: INT:=100;  (* 0:MAN OFF, -1:MAN-ON,
							   -2:KEY-ON, -3:KEY-OFF, -4:DAY, -5:NIGHT,
							   N>0:Nsec-TIMER *)
	CtrlTrig		: BOOL; (* Trigger for timer start *)
	CtrlKey			: BOOL; (* External KEY control input *)
	CtrlSens		: BOOL; (* External dark sensor input [1:Dark] *)
	CtrlExton		: BOOL; (* External forced activation *)
	(* Physical inputs *)
	REL_ST			: BOOL; (* Status feedback *)
	REL_V			: WORD; (* [E-1 V] Voltage *)
	REL_A			: WORD; (* [E-1 A] Current *)
	REL_ALM			: WORD; (* Error status [0:OK, 1:Disconnected, 2:LoadLOW, 3:LoadHIGH, 4:Overload, 5:ControlFAIL] *)
	REL_TEMP		: INT;  (* [E-1 °C] Temperature *)
	REL_TON			: DWORD;(* [sec] External working time counter *)  
	(* Persistent *)(*
	WORKINGTIME		: POINTER TO DWORD; (* [sec] Internal working time counter *)
	POWERONCYCLES	: POINTER TO DWORD; (* Internal counter of power-on cycles *)
	ENERGYCOUNTER	: POINTER TO DWORD; (* [E-1 kWh] Internal energy counter *)
	ENERGYCOUNTER_T : POINTER TO DWORD; (* Temporary energy in E-2*Wsec *)*)
	PressKeyVisuOn	: BOOL := 0;
	PressKeyVisuOff	: BOOL := 0;
END_VAR
VAR_IN_OUT
//VAR_OUTPUT RETAIN PERSISTENT
	
	WORKINGTIME		: DWORD; (* [sec] Internal working time counter *)
	POWERONCYCLES	: DWORD; (* Internal counter of power-on cycles *)
	ENERGYCOUNTER	: DWORD; (* [E-1 kWh] Internal energy counter *)
	ENERGYCOUNTER_T : DWORD; (* Temporary energy in E-2*Wsec *)
END_VAR
VAR_OUTPUT
	(* Physical outputs *)
	REL_EN			: BOOL;	(* Control output *)
	(* Status *)
	Status_Log		: BYTE;
	Status_Vis 		: DWORD;
END_VAR
VAR
	TickTimer		: TON := ( PT:=T#1S );
	TrigTimer		: TOF ;
	sREL_EN			: FLT_EVENT;
	sREL_ALM		: WORD:=16#FFFF;
	chkREL_ST		: FLT_TIME := ( TTAP:=T#20S, INITEV:=FALSE );
	
END_VAR

(* Trig timer *)
TrigTimer.PT:=TIME_LUX_DEF;
TrigTimer(IN:= CtrlTrig);

IF TrigTimer.Q THEN 
	//LUX_LIST[ID] := FALSE;
	LuxOutput_ASI[ID] := FALSE;
	//LUXM_46:=FALSE;	
	ELSE
		//LUX_LIST[ID] := TRUE;
		LuxOutput_ASI[ID] := TRUE;
		//LUXM_46:=TRUE;	
END_IF
RETURN;

